Universal Robots URScript: etalement_vINIT.script

# UR5 - Protocole etalement cosmetique
# Genere automatiquement par ur5_etalement.py
# IMPORTANT : calibrer ROBOT_X_ORIGIN, ROBOT_Y_ORIGIN, ROBOT_Z_SURFACE avant execution

# --- Ancre globale du repere de travail ---
# P_ANCHOR_OLD : ancre nominale de la trajectoire originale (NE PAS MODIFIER)
# P_REF        : ancre cible. Modifier cette ligne pour relocaliser toute la zone d'etalement.
global P_ANCHOR_OLD = p[0.2,   -0.335, 0.05, 3.14159, 0.0, 0.0]
global P_REF        = p[-0.011, 0.6,   -0.3, 0.0, -3.1416, 0.0]


#TODO 5- Le nombre de lignes de code dans le script généré pour le robot UR5 dans UR5_etalementv6.py, est potentiellement trop élevé. Ce nombre de ligne de code dans le script est directement lié à la discretisation des cercles avec leur translation et la commande de force lors de chaque déplacement du robot UR5 sur le plan X-Y. Une option serait d'utiliser une fonction dans le robot UR5 pour réaliser des cercles avec translation sans l'utilisation de points avec la fonction movel tout en conservant en tout temps une commande pour 6N perpendiculaire au plan. Propose un plan pour réaliser ces fonctions dédiées. L'option des points de discrétisation doit demeurer. Il faut ajouter une option pour utiliser une fonction cercle+translation avec une sélection sous les figures.

# --- Vitesses (m/s) par phase ---
global V_APPROACH = 0.3
global V_CONTACT  = 0.05
global V_CIRC     = 0.0360
global V_RECT     = 0.0800
global V_INIT     = 0.5

# --- Accelerations (m/s^2) par phase ---
global A_DEFAULT  = 0.8
global A_INIT     = 1.2

# --- Facteurs multiplicateurs globaux ---
# 1.0 = nominal. Reduire SPEED_FACTOR pour mise au point.
global SPEED_FACTOR = 1.0
global ACCEL_FACTOR = 1.0

def T(p_orig):
  return pose_trans(P_REF, pose_trans(pose_inv(P_ANCHOR_OLD), p_orig))
end

def cycle_1():
  # --- Cycle 1 - Circulaire (0deg) ---
  movel(T(p[0.196464, -0.310607, 0.060000, 3.14159, 0.0, 0.0]), a=A_DEFAULT*ACCEL_FACTOR, v=V_APPROACH*SPEED_FACTOR)
  movel(T(p[0.196464, -0.310607, 0.050000, 3.14159, 0.0, 0.0]), a=A_DEFAULT*ACCEL_FACTOR, v=V_CONTACT*SPEED_FACTOR)
  force_mode(get_actual_tcp_pose(), [0, 0, 1, 0, 0, 0], [0, 0, -6.0, 0, 0, 0], 2, [0.002, 0.002, 0.04, 0.35, 0.35, 0.35])
  movel(T(p[0.198247, -0.304185, 0.050000, 3.14159, 0.0, 0.0]), a=A_DEFAULT*ACCEL_FACTOR, v=V_CIRC*SPEED_FACTOR, r=0.002)
  movel(T(p[0.206814, -0.307177, 0.050000, 3.14159, 0.0, 0.0]), a=A_DEFAULT*ACCEL_FACTOR, v=V_CIRC*SPEED_FACTOR, r=0.002)
  movel(T(p[0.205001, -0.315356, 0.050000, 3.14159, 0.0, 0.0]), a=A_DEFAULT*ACCEL_FACTOR, v=V_CIRC*SPEED_FACTOR, r=0.002)
  movel(T(p[0.199733, -0.312459, 0.050000, 3.14159, 0.0, 0.0]), a=A_DEFAULT*ACCEL_FACTOR, v=V_CIRC*SPEED_FACTOR, r=0.002)
  movel(T(p[0.206632, -0.307954, 0.050000, 3.14159, 0.0, 0.0]), a=A_DEFAULT*ACCEL_FACTOR, v=V_CIRC*SPEED_FACTOR, r=0.002)
  movel(T(p[0.211681, -0.315756, 0.050000, 3.14159, 0.0, 0.0]), a=A_DEFAULT*ACCEL_FACTOR, v=V_CIRC*SPEED_FACTOR, r=0.002)
  movel(T(p[0.205611, -0.319527, 0.050000, 3.14159, 0.0, 0.0]), a=A_DEFAULT*ACCEL_FACTOR, v=V_CIRC*SPEED_FACTOR, r=0.002)
  movel(T(p[0.205535, -0.313103, 0.050000, 3.14159, 0.0, 0.0]), a=A_DEFAULT*ACCEL_FACTOR, v=V_CIRC*SPEED_FACTOR, r=0.002)
  movel(T(p[0.214388, -0.314433, 0.050000, 3.14159, 0.0, 0.0]), a=A_DEFAULT*ACCEL_FACTOR, v=V_CIRC*SPEED_FACTOR, r=0.002)
  movel(T(p[0.213984, -0.323127, 0.050000, 3.14159, 0.0, 0.0]), a=A_DEFAULT*ACCEL_FACTOR, v=V_CIRC*SPEED_FACTOR, r=0.002)
  movel(T(p[0.208033, -0.321374, 0.050000, 3.14159, 0.0, 0.0]), a=A_DEFAULT*ACCEL_FACTOR, v=V_CIRC*SPEED_FACTOR, r=0.002)
  movel(T(p[0.213367, -0.316077, 0.050000, 3.14159, 0.0, 0.0]), a=A_DEFAULT*ACCEL_FACTOR, v=V_CIRC*SPEED_FACTOR, r=0.002)
  movel(T(p[0.220124, -0.322521, 0.050000, 3.14159, 0.0, 0.0]), a=A_DEFAULT*ACCEL_FACTOR, v=V_CIRC*SPEED_FACTOR, r=0.002)
  movel(T(p[0.215077, -0.328218, 0.050000, 3.14159, 0.0, 0.0]), a=A_DEFAULT*ACCEL_FACTOR, v=V_CIRC*SPEED_FACTOR, r=0.002)
  movel(T(p[0.212920, -0.322447, 0.050000, 3.14159, 0.0, 0.0]), a=A_DEFAULT*ACCEL_FACTOR, v=V_CIRC*SPEED_FACTOR, r=0.002)
  movel(T(p[0.221510, -0.321613, 0.050000, 3.14159, 0.0, 0.0]), a=A_DEFAULT*ACCEL_FACTOR, v=V_CIRC*SPEED_FACTOR, r=0.002)
  movel(T(p[0.223283, -0.330444, 0.050000, 3.14159, 0.0, 0.0]), a=A_DEFAULT*ACCEL_FACTOR, v=V_CIRC*SPEED_FACTOR, r=0.002)
  movel(T(p[0.216799, -0.330806, 0.050000, 3.14159, 0.0, 0.0]), a=A_DEFAULT*ACCEL_FACTOR, v=V_CIRC*SPEED_FACTOR, r=0.002)
  movel(T(p[0.220152, -0.324598, 0.050000, 3.14159, 0.0, 0.0]), a=A_DEFAULT*ACCEL_FACTOR, v=V_CIRC*SPEED_FACTOR, r=0.002)
  movel(T(p[0.228165, -0.329259, 0.050000, 3.14159, 0.0, 0.0]), a=A_DEFAULT*ACCEL_FACTOR, v=V_CIRC*SPEED_FACTOR, r=0.002)
  movel(T(p[0.224257, -0.340672, 0.050000, 3.14159, 0.0, 0.0]), a=A_DEFAULT*ACCEL_FACTOR, v=V_CIRC*SPEED_FACTOR, r=0.002)
  movel(T(p[0.224298, -0.337927, 0.050000, 3.14159, 0.0, 0.0]), a=A_DEFAULT*ACCEL_FACTOR, v=V_CIRC*SPEED_FACTOR, r=0.002)
  movel(T(p[0.210179, -0.336950, 0.050000, 3.14159, 0.0, 0.0]), a=A_DEFAULT*ACCEL_FACTOR, v=V_CIRC*SPEED_FACTOR, r=0.002)
  movel(T(p[0.216700, -0.335572, 0.050000, 3.14159, 0.0, 0.0]), a=A_DEFAULT*ACCEL_FACTOR, v=V_CIRC*SPEED_FACTOR, r=0.002)
  movel(T(p[0.214342, -0.342004, 0.050000, 3.14159, 0.0, 0.0]), a=A_DEFAULT*ACCEL_FACTOR, v=V_CIRC*SPEED_FACTOR, r=0.002)
  movel(T(p[0.205926, -0.338276, 0.050000, 3.14159, 0.0, 0.0]), a=A_DEFAULT*ACCEL_FACTOR, v=V_CIRC*SPEED_FACTOR, r=0.002)
  movel(T(p[0.208605, -0.330451, 0.050000, 3.14159, 0.0, 0.0]), a=A_DEFAULT*ACCEL_FACTOR, v=V_CIRC*SPEED_FACTOR, r=0.002)
  movel(T(p[0.213287, -0.334283, 0.050000, 3.14159, 0.0, 0.0]), a=A_DEFAULT*ACCEL_FACTOR, v=V_CIRC*SPEED_FACTOR, r=0.002)
  movel(T(p[0.206141, -0.337953, 0.050000, 3.14159, 0.0, 0.0]), a=A_DEFAULT*ACCEL_FACTOR, v=V_CIRC*SPEED_FACTOR, r=0.002)
  movel(T(p[0.201316, -0.330024, 0.050000, 3.14159, 0.0, 0.0]), a=A_DEFAULT*ACCEL_FACTOR, v=V_CIRC*SPEED_FACTOR, r=0.002)
  movel(T(p[0.207470, -0.326497, 0.050000, 3.14159, 0.0, 0.0]), a=A_DEFAULT*ACCEL_FACTOR, v=V_CIRC*SPEED_FACTOR, r=0.002)
  movel(T(p[0.207291, -0.332959, 0.050000, 3.14159, 0.0, 0.0]), a=A_DEFAULT*ACCEL_FACTOR, v=V_CIRC*SPEED_FACTOR, r=0.002)
  movel(T(p[0.198448, -0.331369, 0.050000, 3.14159, 0.0, 0.0]), a=A_DEFAULT*ACCEL_FACTOR, v=V_CIRC*SPEED_FACTOR, r=0.002)
  movel(T(p[0.199103, -0.322733, 0.050000, 3.14159, 0.0, 0.0]), a=A_DEFAULT*ACCEL_FACTOR, v=V_CIRC*SPEED_FACTOR, r=0.002)
  movel(T(p[0.204951, -0.324723, 0.050000, 3.14159, 0.0, 0.0]), a=A_DEFAULT*ACCEL_FACTOR, v=V_CIRC*SPEED_FACTOR, r=0.002)
  movel(T(p[0.199404, -0.329877, 0.050000, 3.14159, 0.0, 0.0]), a=A_DEFAULT*ACCEL_FACTOR, v=V_CIRC*SPEED_FACTOR, r=0.002)
  movel(T(p[0.192828, -0.323249, 0.050000, 3.14159, 0.0, 0.0]), a=A_DEFAULT*ACCEL_FACTOR, v=V_CIRC*SPEED_FACTOR, r=0.002)
  movel(T(p[0.198024, -0.317762, 0.050000, 3.14159, 0.0, 0.0]), a=A_DEFAULT*ACCEL_FACTOR, v=V_CIRC*SPEED_FACTOR, r=0.002)
  movel(T(p[0.199946, -0.323641, 0.050000, 3.14159, 0.0, 0.0]), a=A_DEFAULT*ACCEL_FACTOR, v=V_CIRC*SPEED_FACTOR, r=0.002)
  movel(T(p[0.191594, -0.323878, 0.050000, 3.14159, 0.0, 0.0]), a=A_DEFAULT*ACCEL_FACTOR, v=V_CIRC*SPEED_FACTOR, r=0.002)
  movel(T(p[0.184241, -0.319409, 0.050000, 3.14159, 0.0, 0.0]), a=A_DEFAULT*ACCEL_FACTOR, v=V_CIRC*SPEED_FACTOR, r=0.002)
  movel(T(p[0.184896, -0.325887, 0.050000, 3.14159, 0.0, 0.0]), a=A_DEFAULT*ACCEL_FACTOR, v=V_CIRC*SPEED_FACTOR, r=0.002)
  movel(T(p[0.192145, -0.331753, 0.050000, 3.14159, 0.0, 0.0]), a=A_DEFAULT*ACCEL_FACTOR, v=V_CIRC*SPEED_FACTOR, r=0.002)
  movel(T(p[0.187575, -0.338042, 0.050000, 3.14159, 0.0, 0.0]), a=A_DEFAULT*ACCEL_FACTOR, v=V_CIRC*SPEED_FACTOR, r=0.002)
  movel(T(p[0.184751, -0.332632, 0.050000, 3.14159, 0.0, 0.0]), a=A_DEFAULT*ACCEL_FACTOR, v=V_CIRC*SPEED_FACTOR, r=0.002)
  movel(T(p[0.193108, -0.331077, 0.050000, 3.14159, 0.0, 0.0]), a=A_DEFAULT*ACCEL_FACTOR, v=V_CIRC*SPEED_FACTOR, r=0.002)
  movel(T(p[0.195634, -0.339809, 0.050000, 3.14159, 0.0, 0.0]), a=A_DEFAULT*ACCEL_FACTOR, v=V_CIRC*SPEED_FACTOR, r=0.002)
  movel(T(p[0.189108, -0.340929, 0.050000, 3.14159, 0.0, 0.0]), a=A_DEFAULT*ACCEL_FACTOR, v=V_CIRC*SPEED_FACTOR, r=0.002)
  movel(T(p[0.191723, -0.334542, 0.050000, 3.14159, 0.0, 0.0]), a=A_DEFAULT*ACCEL_FACTOR, v=V_CIRC*SPEED_FACTOR, r=0.002)
  movel(T(p[0.200047, -0.338511, 0.050000, 3.14159, 0.0, 0.0]), a=A_DEFAULT*ACCEL_FACTOR, v=V_CIRC*SPEED_FACTOR, r=0.002)
  movel(T(p[0.197147, -0.346203, 0.050000, 3.14159, 0.0, 0.0]), a=A_DEFAULT*ACCEL_FACTOR, v=V_CIRC*SPEED_FACTOR, r=0.002)
  movel(T(p[0.192637, -0.342178, 0.050000, 3.14159, 0.0, 0.0]), a=A_DEFAULT*ACCEL_FACTOR, v=V_CIRC*SPEED_FACTOR, r=0.002)
  movel(T(p[0.199941, -0.338712, 0.050000, 3.14159, 0.0, 0.0]), a=A_DEFAULT*ACCEL_FACTOR, v=V_CIRC*SPEED_FACTOR, r=0.002)
  movel(T(p[0.204537, -0.346760, 0.050000, 3.14159, 0.0, 0.0]), a=A_DEFAULT*ACCEL_FACTOR, v=V_CIRC*SPEED_FACTOR, r=0.002)
  movel(T(p[0.198308, -0.350040, 0.050000, 3.14159, 0.0, 0.0]), a=A_DEFAULT*ACCEL_FACTOR, v=V_CIRC*SPEED_FACTOR, r=0.002)
  movel(T(p[0.198743, -0.343549, 0.050000, 3.14159, 0.0, 0.0]), a=A_DEFAULT*ACCEL_FACTOR, v=V_CIRC*SPEED_FACTOR, r=0.002)
  movel(T(p[0.207568, -0.345396, 0.050000, 3.14159, 0.0, 0.0]), a=A_DEFAULT*ACCEL_FACTOR, v=V_CIRC*SPEED_FACTOR, r=0.002)
  movel(T(p[0.206662, -0.353966, 0.050000, 3.14159, 0.0, 0.0]), a=A_DEFAULT*ACCEL_FACTOR, v=V_CIRC*SPEED_FACTOR, r=0.002)
  movel(T(p[0.210965, -0.358063, 0.050000, 3.14159, 0.0, 0.0]), a=A_DEFAULT*ACCEL_FACTOR, v=V_CIRC*SPEED_FACTOR, r=0.002)
  movel(T(p[0.197831, -0.356868, 0.050000, 3.14159, 0.0, 0.0]), a=A_DEFAULT*ACCEL_FACTOR, v=V_CIRC*SPEED_FACTOR, r=0.002)
  movel(T(p[0.197313, -0.354239, 0.050000, 3.14159, 0.0, 0.0]), a=A_DEFAULT*ACCEL_FACTOR, v=V_CIRC*SPEED_FACTOR, r=0.002)
  movel(T(p[0.197882, -0.360567, 0.050000, 3.14159, 0.0, 0.0]), a=A_DEFAULT*ACCEL_FACTOR, v=V_CIRC*SPEED_FACTOR, r=0.002)
  movel(T(p[0.189034, -0.359736, 0.050000, 3.14159, 0.0, 0.0]), a=A_DEFAULT*ACCEL_FACTOR, v=V_CIRC*SPEED_FACTOR, r=0.002)
  movel(T(p[0.188944, -0.350957, 0.050000, 3.14159, 0.0, 0.0]), a=A_DEFAULT*ACCEL_FACTOR, v=V_CIRC*SPEED_FACTOR, r=0.002)
  movel(T(p[0.195069, -0.352240, 0.050000, 3.14159, 0.0, 0.0]), a=A_DEFAULT*ACCEL_FACTOR, v=V_CIRC*SPEED_FACTOR, r=0.002)
  movel(T(p[0.190166, -0.357795, 0.050000, 3.14159, 0.0, 0.0]), a=A_DEFAULT*ACCEL_FACTOR, v=V_CIRC*SPEED_FACTOR, r=0.002)
  movel(T(p[0.183077, -0.351727, 0.050000, 3.14159, 0.0, 0.0]), a=A_DEFAULT*ACCEL_FACTOR, v=V_CIRC*SPEED_FACTOR, r=0.002)
  movel(T(p[0.187816, -0.345635, 0.050000, 3.14159, 0.0, 0.0]), a=A_DEFAULT*ACCEL_FACTOR, v=V_CIRC*SPEED_FACTOR, r=0.002)
  movel(T(p[0.190418, -0.351174, 0.050000, 3.14159, 0.0, 0.0]), a=A_DEFAULT*ACCEL_FACTOR, v=V_CIRC*SPEED_FACTOR, r=0.002)
  movel(T(p[0.181973, -0.352487, 0.050000, 3.14159, 0.0, 0.0]), a=A_DEFAULT*ACCEL_FACTOR, v=V_CIRC*SPEED_FACTOR, r=0.002)
  movel(T(p[0.179702, -0.343713, 0.050000, 3.14159, 0.0, 0.0]), a=A_DEFAULT*ACCEL_FACTOR, v=V_CIRC*SPEED_FACTOR, r=0.002)
  movel(T(p[0.186221, -0.342851, 0.050000, 3.14159, 0.0, 0.0]), a=A_DEFAULT*ACCEL_FACTOR, v=V_CIRC*SPEED_FACTOR, r=0.002)
  movel(T(p[0.183355, -0.349185, 0.050000, 3.14159, 0.0, 0.0]), a=A_DEFAULT*ACCEL_FACTOR, v=V_CIRC*SPEED_FACTOR, r=0.002)
  movel(T(p[0.175128, -0.344978, 0.050000, 3.14159, 0.0, 0.0]), a=A_DEFAULT*ACCEL_FACTOR, v=V_CIRC*SPEED_FACTOR, r=0.002)
  movel(T(p[0.178246, -0.337425, 0.050000, 3.14159, 0.0, 0.0]), a=A_DEFAULT*ACCEL_FACTOR, v=V_CIRC*SPEED_FACTOR, r=0.002)
  movel(T(p[0.182578, -0.341638, 0.050000, 3.14159, 0.0, 0.0]), a=A_DEFAULT*ACCEL_FACTOR, v=V_CIRC*SPEED_FACTOR, r=0.002)
  movel(T(p[0.175123, -0.344896, 0.050000, 3.14159, 0.0, 0.0]), a=A_DEFAULT*ACCEL_FACTOR, v=V_CIRC*SPEED_FACTOR, r=0.002)
  movel(T(p[0.171025, -0.336323, 0.050000, 3.14159, 0.0, 0.0]), a=A_DEFAULT*ACCEL_FACTOR, v=V_CIRC*SPEED_FACTOR, r=0.002)
  movel(T(p[0.177378, -0.333966, 0.050000, 3.14159, 0.0, 0.0]), a=A_DEFAULT*ACCEL_FACTOR, v=V_CIRC*SPEED_FACTOR, r=0.002)
  movel(T(p[0.176172, -0.340413, 0.050000, 3.14159, 0.0, 0.0]), a=A_DEFAULT*ACCEL_FACTOR, v=V_CIRC*SPEED_FACTOR, r=0.002)
  movel(T(p[0.167489, -0.337986, 0.050000, 3.14159, 0.0, 0.0]), a=A_DEFAULT*ACCEL_FACTOR, v=V_CIRC*SPEED_FACTOR, r=0.002)
  end_force_mode()
  movel(T(p[0.168180, -0.338891, 0.060000, 3.14159, 0.0, 0.0]), a=A_DEFAULT*ACCEL_FACTOR, v=V_APPROACH*SPEED_FACTOR)
end

def cycle_2():
  # --- Cycle 2 - Circulaire (90deg) ---
  movel(T(p[0.175251, -0.338891, 0.060000, 3.14159, 0.0, 0.0]), a=A_DEFAULT*ACCEL_FACTOR, v=V_APPROACH*SPEED_FACTOR)
  movel(T(p[0.175251, -0.338891, 0.050000, 3.14159, 0.0, 0.0]), a=A_DEFAULT*ACCEL_FACTOR, v=V_CONTACT*SPEED_FACTOR)
  force_mode(get_actual_tcp_pose(), [0, 0, 1, 0, 0, 0], [0, 0, -6.0, 0, 0, 0], 2, [0.002, 0.002, 0.04, 0.35, 0.35, 0.35])
  movel(T(p[0.168830, -0.337108, 0.050000, 3.14159, 0.0, 0.0]), a=A_DEFAULT*ACCEL_FACTOR, v=V_CIRC*SPEED_FACTOR, r=0.002)
  movel(T(p[0.171822, -0.328542, 0.050000, 3.14159, 0.0, 0.0]), a=A_DEFAULT*ACCEL_FACTOR, v=V_CIRC*SPEED_FACTOR, r=0.002)
  movel(T(p[0.180001, -0.330354, 0.050000, 3.14159, 0.0, 0.0]), a=A_DEFAULT*ACCEL_FACTOR, v=V_CIRC*SPEED_FACTOR, r=0.002)
  movel(T(p[0.177104, -0.335623, 0.050000, 3.14159, 0.0, 0.0]), a=A_DEFAULT*ACCEL_FACTOR, v=V_CIRC*SPEED_FACTOR, r=0.002)
  movel(T(p[0.172599, -0.328723, 0.050000, 3.14159, 0.0, 0.0]), a=A_DEFAULT*ACCEL_FACTOR, v=V_CIRC*SPEED_FACTOR, r=0.002)
  movel(T(p[0.180400, -0.323674, 0.050000, 3.14159, 0.0, 0.0]), a=A_DEFAULT*ACCEL_FACTOR, v=V_CIRC*SPEED_FACTOR, r=0.002)
  movel(T(p[0.184171, -0.329744, 0.050000, 3.14159, 0.0, 0.0]), a=A_DEFAULT*ACCEL_FACTOR, v=V_CIRC*SPEED_FACTOR, r=0.002)
  movel(T(p[0.177747, -0.329820, 0.050000, 3.14159, 0.0, 0.0]), a=A_DEFAULT*ACCEL_FACTOR, v=V_CIRC*SPEED_FACTOR, r=0.002)
  movel(T(p[0.179078, -0.320967, 0.050000, 3.14159, 0.0, 0.0]), a=A_DEFAULT*ACCEL_FACTOR, v=V_CIRC*SPEED_FACTOR, r=0.002)
  movel(T(p[0.187771, -0.321372, 0.050000, 3.14159, 0.0, 0.0]), a=A_DEFAULT*ACCEL_FACTOR, v=V_CIRC*SPEED_FACTOR, r=0.002)
  movel(T(p[0.186018, -0.327322, 0.050000, 3.14159, 0.0, 0.0]), a=A_DEFAULT*ACCEL_FACTOR, v=V_CIRC*SPEED_FACTOR, r=0.002)
  movel(T(p[0.180721, -0.321988, 0.050000, 3.14159, 0.0, 0.0]), a=A_DEFAULT*ACCEL_FACTOR, v=V_CIRC*SPEED_FACTOR, r=0.002)
  movel(T(p[0.187165, -0.315232, 0.050000, 3.14159, 0.0, 0.0]), a=A_DEFAULT*ACCEL_FACTOR, v=V_CIRC*SPEED_FACTOR, r=0.002)
  movel(T(p[0.192862, -0.320278, 0.050000, 3.14159, 0.0, 0.0]), a=A_DEFAULT*ACCEL_FACTOR, v=V_CIRC*SPEED_FACTOR, r=0.002)
  movel(T(p[0.187092, -0.322436, 0.050000, 3.14159, 0.0, 0.0]), a=A_DEFAULT*ACCEL_FACTOR, v=V_CIRC*SPEED_FACTOR, r=0.002)
  movel(T(p[0.186258, -0.313845, 0.050000, 3.14159, 0.0, 0.0]), a=A_DEFAULT*ACCEL_FACTOR, v=V_CIRC*SPEED_FACTOR, r=0.002)
  movel(T(p[0.195089, -0.312072, 0.050000, 3.14159, 0.0, 0.0]), a=A_DEFAULT*ACCEL_FACTOR, v=V_CIRC*SPEED_FACTOR, r=0.002)
  movel(T(p[0.195450, -0.318556, 0.050000, 3.14159, 0.0, 0.0]), a=A_DEFAULT*ACCEL_FACTOR, v=V_CIRC*SPEED_FACTOR, r=0.002)
  movel(T(p[0.189243, -0.315204, 0.050000, 3.14159, 0.0, 0.0]), a=A_DEFAULT*ACCEL_FACTOR, v=V_CIRC*SPEED_FACTOR, r=0.002)
  movel(T(p[0.193904, -0.307191, 0.050000, 3.14159, 0.0, 0.0]), a=A_DEFAULT*ACCEL_FACTOR, v=V_CIRC*SPEED_FACTOR, r=0.002)
  movel(T(p[0.205317, -0.311098, 0.050000, 3.14159, 0.0, 0.0]), a=A_DEFAULT*ACCEL_FACTOR, v=V_CIRC*SPEED_FACTOR, r=0.002)
  movel(T(p[0.202572, -0.311057, 0.050000, 3.14159, 0.0, 0.0]), a=A_DEFAULT*ACCEL_FACTOR, v=V_CIRC*SPEED_FACTOR, r=0.002)
  movel(T(p[0.201595, -0.325177, 0.050000, 3.14159, 0.0, 0.0]), a=A_DEFAULT*ACCEL_FACTOR, v=V_CIRC*SPEED_FACTOR, r=0.002)
  movel(T(p[0.200216, -0.318655, 0.050000, 3.14159, 0.0, 0.0]), a=A_DEFAULT*ACCEL_FACTOR, v=V_CIRC*SPEED_FACTOR, r=0.002)
  movel(T(p[0.206648, -0.321014, 0.050000, 3.14159, 0.0, 0.0]), a=A_DEFAULT*ACCEL_FACTOR, v=V_CIRC*SPEED_FACTOR, r=0.002)
  movel(T(p[0.202920, -0.329430, 0.050000, 3.14159, 0.0, 0.0]), a=A_DEFAULT*ACCEL_FACTOR, v=V_CIRC*SPEED_FACTOR, r=0.002)
  movel(T(p[0.195096, -0.326750, 0.050000, 3.14159, 0.0, 0.0]), a=A_DEFAULT*ACCEL_FACTOR, v=V_CIRC*SPEED_FACTOR, r=0.002)
  movel(T(p[0.198928, -0.322069, 0.050000, 3.14159, 0.0, 0.0]), a=A_DEFAULT*ACCEL_FACTOR, v=V_CIRC*SPEED_FACTOR, r=0.002)
  movel(T(p[0.202597, -0.329214, 0.050000, 3.14159, 0.0, 0.0]), a=A_DEFAULT*ACCEL_FACTOR, v=V_CIRC*SPEED_FACTOR, r=0.002)
  movel(T(p[0.194669, -0.334039, 0.050000, 3.14159, 0.0, 0.0]), a=A_DEFAULT*ACCEL_FACTOR, v=V_CIRC*SPEED_FACTOR, r=0.002)
  movel(T(p[0.191141, -0.327885, 0.050000, 3.14159, 0.0, 0.0]), a=A_DEFAULT*ACCEL_FACTOR, v=V_CIRC*SPEED_FACTOR, r=0.002)
  movel(T(p[0.197604, -0.328064, 0.050000, 3.14159, 0.0, 0.0]), a=A_DEFAULT*ACCEL_FACTOR, v=V_CIRC*SPEED_FACTOR, r=0.002)
  movel(T(p[0.196014, -0.336907, 0.050000, 3.14159, 0.0, 0.0]), a=A_DEFAULT*ACCEL_FACTOR, v=V_CIRC*SPEED_FACTOR, r=0.002)
  movel(T(p[0.187378, -0.336252, 0.050000, 3.14159, 0.0, 0.0]), a=A_DEFAULT*ACCEL_FACTOR, v=V_CIRC*SPEED_FACTOR, r=0.002)
  movel(T(p[0.189368, -0.330404, 0.050000, 3.14159, 0.0, 0.0]), a=A_DEFAULT*ACCEL_FACTOR, v=V_CIRC*SPEED_FACTOR, r=0.002)
  movel(T(p[0.194522, -0.335951, 0.050000, 3.14159, 0.0, 0.0]), a=A_DEFAULT*ACCEL_FACTOR, v=V_CIRC*SPEED_FACTOR, r=0.002)
  movel(T(p[0.187894, -0.342528, 0.050000, 3.14159, 0.0, 0.0]), a=A_DEFAULT*ACCEL_FACTOR, v=V_CIRC*SPEED_FACTOR, r=0.002)
  movel(T(p[0.182406, -0.337332, 0.050000, 3.14159, 0.0, 0.0]), a=A_DEFAULT*ACCEL_FACTOR, v=V_CIRC*SPEED_FACTOR, r=0.002)
  movel(T(p[0.188285, -0.335410, 0.050000, 3.14159, 0.0, 0.0]), a=A_DEFAULT*ACCEL_FACTOR, v=V_CIRC*SPEED_FACTOR, r=0.002)
  movel(T(p[0.188522, -0.343761, 0.050000, 3.14159, 0.0, 0.0]), a=A_DEFAULT*ACCEL_FACTOR, v=V_CIRC*SPEED_FACTOR, r=0.002)
  movel(T(p[0.184054, -0.351115, 0.050000, 3.14159, 0.0, 0.0]), a=A_DEFAULT*ACCEL_FACTOR, v=V_CIRC*SPEED_FACTOR, r=0.002)
  movel(T(p[0.190532, -0.350459, 0.050000, 3.14159, 0.0, 0.0]), a=A_DEFAULT*ACCEL_FACTOR, v=V_CIRC*SPEED_FACTOR, r=0.002)
  movel(T(p[0.196398, -0.343210, 0.050000, 3.14159, 0.0, 0.0]), a=A_DEFAULT*ACCEL_FACTOR, v=V_CIRC*SPEED_FACTOR, r=0.002)
  movel(T(p[0.202686, -0.347780, 0.050000, 3.14159, 0.0, 0.0]), a=A_DEFAULT*ACCEL_FACTOR, v=V_CIRC*SPEED_FACTOR, r=0.002)
  movel(T(p[0.197277, -0.350604, 0.050000, 3.14159, 0.0, 0.0]), a=A_DEFAULT*ACCEL_FACTOR, v=V_CIRC*SPEED_FACTOR, r=0.002)
  movel(T(p[0.195721, -0.342248, 0.050000, 3.14159, 0.0, 0.0]), a=A_DEFAULT*ACCEL_FACTOR, v=V_CIRC*SPEED_FACTOR, r=0.002)
  movel(T(p[0.204454, -0.339722, 0.050000, 3.14159, 0.0, 0.0]), a=A_DEFAULT*ACCEL_FACTOR, v=V_CIRC*SPEED_FACTOR, r=0.002)
  movel(T(p[0.205574, -0.346247, 0.050000, 3.14159, 0.0, 0.0]), a=A_DEFAULT*ACCEL_FACTOR, v=V_CIRC*SPEED_FACTOR, r=0.002)
  movel(T(p[0.199187, -0.343633, 0.050000, 3.14159, 0.0, 0.0]), a=A_DEFAULT*ACCEL_FACTOR, v=V_CIRC*SPEED_FACTOR, r=0.002)
  movel(T(p[0.203156, -0.335308, 0.050000, 3.14159, 0.0, 0.0]), a=A_DEFAULT*ACCEL_FACTOR, v=V_CIRC*SPEED_FACTOR, r=0.002)
  movel(T(p[0.210848, -0.338209, 0.050000, 3.14159, 0.0, 0.0]), a=A_DEFAULT*ACCEL_FACTOR, v=V_CIRC*SPEED_FACTOR, r=0.002)
  movel(T(p[0.206823, -0.342718, 0.050000, 3.14159, 0.0, 0.0]), a=A_DEFAULT*ACCEL_FACTOR, v=V_CIRC*SPEED_FACTOR, r=0.002)
  movel(T(p[0.203357, -0.335414, 0.050000, 3.14159, 0.0, 0.0]), a=A_DEFAULT*ACCEL_FACTOR, v=V_CIRC*SPEED_FACTOR, r=0.002)
  movel(T(p[0.211404, -0.330819, 0.050000, 3.14159, 0.0, 0.0]), a=A_DEFAULT*ACCEL_FACTOR, v=V_CIRC*SPEED_FACTOR, r=0.002)
  movel(T(p[0.214684, -0.337047, 0.050000, 3.14159, 0.0, 0.0]), a=A_DEFAULT*ACCEL_FACTOR, v=V_CIRC*SPEED_FACTOR, r=0.002)
  movel(T(p[0.208193, -0.336612, 0.050000, 3.14159, 0.0, 0.0]), a=A_DEFAULT*ACCEL_FACTOR, v=V_CIRC*SPEED_FACTOR, r=0.002)
  movel(T(p[0.210040, -0.327787, 0.050000, 3.14159, 0.0, 0.0]), a=A_DEFAULT*ACCEL_FACTOR, v=V_CIRC*SPEED_FACTOR, r=0.002)
  movel(T(p[0.218611, -0.328693, 0.050000, 3.14159, 0.0, 0.0]), a=A_DEFAULT*ACCEL_FACTOR, v=V_CIRC*SPEED_FACTOR, r=0.002)
  movel(T(p[0.222707, -0.324390, 0.050000, 3.14159, 0.0, 0.0]), a=A_DEFAULT*ACCEL_FACTOR, v=V_CIRC*SPEED_FACTOR, r=0.002)
  movel(T(p[0.221512, -0.337524, 0.050000, 3.14159, 0.0, 0.0]), a=A_DEFAULT*ACCEL_FACTOR, v=V_CIRC*SPEED_FACTOR, r=0.002)
  movel(T(p[0.218884, -0.338042, 0.050000, 3.14159, 0.0, 0.0]), a=A_DEFAULT*ACCEL_FACTOR, v=V_CIRC*SPEED_FACTOR, r=0.002)
  movel(T(p[0.225211, -0.337474, 0.050000, 3.14159, 0.0, 0.0]), a=A_DEFAULT*ACCEL_FACTOR, v=V_CIRC*SPEED_FACTOR, r=0.002)
  movel(T(p[0.224381, -0.346321, 0.050000, 3.14159, 0.0, 0.0]), a=A_DEFAULT*ACCEL_FACTOR, v=V_CIRC*SPEED_FACTOR, r=0.002)
  movel(T(p[0.215602, -0.346412, 0.050000, 3.14159, 0.0, 0.0]), a=A_DEFAULT*ACCEL_FACTOR, v=V_CIRC*SPEED_FACTOR, r=0.002)
  movel(T(p[0.216885, -0.340286, 0.050000, 3.14159, 0.0, 0.0]), a=A_DEFAULT*ACCEL_FACTOR, v=V_CIRC*SPEED_FACTOR, r=0.002)
  movel(T(p[0.222440, -0.345189, 0.050000, 3.14159, 0.0, 0.0]), a=A_DEFAULT*ACCEL_FACTOR, v=V_CIRC*SPEED_FACTOR, r=0.002)
  movel(T(p[0.216372, -0.352279, 0.050000, 3.14159, 0.0, 0.0]), a=A_DEFAULT*ACCEL_FACTOR, v=V_CIRC*SPEED_FACTOR, r=0.002)
  movel(T(p[0.210279, -0.347539, 0.050000, 3.14159, 0.0, 0.0]), a=A_DEFAULT*ACCEL_FACTOR, v=V_CIRC*SPEED_FACTOR, r=0.002)
  movel(T(p[0.215819, -0.344937, 0.050000, 3.14159, 0.0, 0.0]), a=A_DEFAULT*ACCEL_FACTOR, v=V_CIRC*SPEED_FACTOR, r=0.002)
  movel(T(p[0.217132, -0.353382, 0.050000, 3.14159, 0.0, 0.0]), a=A_DEFAULT*ACCEL_FACTOR, v=V_CIRC*SPEED_FACTOR, r=0.002)
  movel(T(p[0.208357, -0.355653, 0.050000, 3.14159, 0.0, 0.0]), a=A_DEFAULT*ACCEL_FACTOR, v=V_CIRC*SPEED_FACTOR, r=0.002)
  movel(T(p[0.207495, -0.349134, 0.050000, 3.14159, 0.0, 0.0]), a=A_DEFAULT*ACCEL_FACTOR, v=V_CIRC*SPEED_FACTOR, r=0.002)
  movel(T(p[0.213830, -0.352001, 0.050000, 3.14159, 0.0, 0.0]), a=A_DEFAULT*ACCEL_FACTOR, v=V_CIRC*SPEED_FACTOR, r=0.002)
  movel(T(p[0.209622, -0.360227, 0.050000, 3.14159, 0.0, 0.0]), a=A_DEFAULT*ACCEL_FACTOR, v=V_CIRC*SPEED_FACTOR, r=0.002)
  movel(T(p[0.202070, -0.357109, 0.050000, 3.14159, 0.0, 0.0]), a=A_DEFAULT*ACCEL_FACTOR, v=V_CIRC*SPEED_FACTOR, r=0.002)
  movel(T(p[0.206283, -0.352778, 0.050000, 3.14159, 0.0, 0.0]), a=A_DEFAULT*ACCEL_FACTOR, v=V_CIRC*SPEED_FACTOR, r=0.002)
  movel(T(p[0.209540, -0.360233, 0.050000, 3.14159, 0.0, 0.0]), a=A_DEFAULT*ACCEL_FACTOR, v=V_CIRC*SPEED_FACTOR, r=0.002)
  movel(T(p[0.200968, -0.364330, 0.050000, 3.14159, 0.0, 0.0]), a=A_DEFAULT*ACCEL_FACTOR, v=V_CIRC*SPEED_FACTOR, r=0.002)
  movel(T(p[0.198611, -0.357978, 0.050000, 3.14159, 0.0, 0.0]), a=A_DEFAULT*ACCEL_FACTOR, v=V_CIRC*SPEED_FACTOR, r=0.002)
  movel(T(p[0.205057, -0.359183, 0.050000, 3.14159, 0.0, 0.0]), a=A_DEFAULT*ACCEL_FACTOR, v=V_CIRC*SPEED_FACTOR, r=0.002)
  movel(T(p[0.202631, -0.367866, 0.050000, 3.14159, 0.0, 0.0]), a=A_DEFAULT*ACCEL_FACTOR, v=V_CIRC*SPEED_FACTOR, r=0.002)
  end_force_mode()
  movel(T(p[0.203536, -0.367175, 0.060000, 3.14159, 0.0, 0.0]), a=A_DEFAULT*ACCEL_FACTOR, v=V_APPROACH*SPEED_FACTOR)
end

def cycle_3():
  # --- Cycle 3 - Circulaire (0deg) ---
  movel(T(p[0.196464, -0.310607, 0.060000, 3.14159, 0.0, 0.0]), a=A_DEFAULT*ACCEL_FACTOR, v=V_APPROACH*SPEED_FACTOR)
  movel(T(p[0.196464, -0.310607, 0.050000, 3.14159, 0.0, 0.0]), a=A_DEFAULT*ACCEL_FACTOR, v=V_CONTACT*SPEED_FACTOR)
  force_mode(get_actual_tcp_pose(), [0, 0, 1, 0, 0, 0], [0, 0, -6.0, 0, 0, 0], 2, [0.002, 0.002, 0.04, 0.35, 0.35, 0.35])
  movel(T(p[0.198247, -0.304185, 0.050000, 3.14159, 0.0, 0.0]), a=A_DEFAULT*ACCEL_FACTOR, v=V_CIRC*SPEED_FACTOR, r=0.002)
  movel(T(p[0.206814, -0.307177, 0.050000, 3.14159, 0.0, 0.0]), a=A_DEFAULT*ACCEL_FACTOR, v=V_CIRC*SPEED_FACTOR, r=0.002)
  movel(T(p[0.205001, -0.315356, 0.050000, 3.14159, 0.0, 0.0]), a=A_DEFAULT*ACCEL_FACTOR, v=V_CIRC*SPEED_FACTOR, r=0.002)
  movel(T(p[0.199733, -0.312459, 0.050000, 3.14159, 0.0, 0.0]), a=A_DEFAULT*ACCEL_FACTOR, v=V_CIRC*SPEED_FACTOR, r=0.002)
  movel(T(p[0.206632, -0.307954, 0.050000, 3.14159, 0.0, 0.0]), a=A_DEFAULT*ACCEL_FACTOR, v=V_CIRC*SPEED_FACTOR, r=0.002)
  movel(T(p[0.211681, -0.315756, 0.050000, 3.14159, 0.0, 0.0]), a=A_DEFAULT*ACCEL_FACTOR, v=V_CIRC*SPEED_FACTOR, r=0.002)
  movel(T(p[0.205611, -0.319527, 0.050000, 3.14159, 0.0, 0.0]), a=A_DEFAULT*ACCEL_FACTOR, v=V_CIRC*SPEED_FACTOR, r=0.002)
  movel(T(p[0.205535, -0.313103, 0.050000, 3.14159, 0.0, 0.0]), a=A_DEFAULT*ACCEL_FACTOR, v=V_CIRC*SPEED_FACTOR, r=0.002)
  movel(T(p[0.214388, -0.314433, 0.050000, 3.14159, 0.0, 0.0]), a=A_DEFAULT*ACCEL_FACTOR, v=V_CIRC*SPEED_FACTOR, r=0.002)
  movel(T(p[0.213984, -0.323127, 0.050000, 3.14159, 0.0, 0.0]), a=A_DEFAULT*ACCEL_FACTOR, v=V_CIRC*SPEED_FACTOR, r=0.002)
  movel(T(p[0.208033, -0.321374, 0.050000, 3.14159, 0.0, 0.0]), a=A_DEFAULT*ACCEL_FACTOR, v=V_CIRC*SPEED_FACTOR, r=0.002)
  movel(T(p[0.213367, -0.316077, 0.050000, 3.14159, 0.0, 0.0]), a=A_DEFAULT*ACCEL_FACTOR, v=V_CIRC*SPEED_FACTOR, r=0.002)
  movel(T(p[0.220124, -0.322521, 0.050000, 3.14159, 0.0, 0.0]), a=A_DEFAULT*ACCEL_FACTOR, v=V_CIRC*SPEED_FACTOR, r=0.002)
  movel(T(p[0.215077, -0.328218, 0.050000, 3.14159, 0.0, 0.0]), a=A_DEFAULT*ACCEL_FACTOR, v=V_CIRC*SPEED_FACTOR, r=0.002)
  movel(T(p[0.212920, -0.322447, 0.050000, 3.14159, 0.0, 0.0]), a=A_DEFAULT*ACCEL_FACTOR, v=V_CIRC*SPEED_FACTOR, r=0.002)
  movel(T(p[0.221510, -0.321613, 0.050000, 3.14159, 0.0, 0.0]), a=A_DEFAULT*ACCEL_FACTOR, v=V_CIRC*SPEED_FACTOR, r=0.002)
  movel(T(p[0.223283, -0.330444, 0.050000, 3.14159, 0.0, 0.0]), a=A_DEFAULT*ACCEL_FACTOR, v=V_CIRC*SPEED_FACTOR, r=0.002)
  movel(T(p[0.216799, -0.330806, 0.050000, 3.14159, 0.0, 0.0]), a=A_DEFAULT*ACCEL_FACTOR, v=V_CIRC*SPEED_FACTOR, r=0.002)
  movel(T(p[0.220152, -0.324598, 0.050000, 3.14159, 0.0, 0.0]), a=A_DEFAULT*ACCEL_FACTOR, v=V_CIRC*SPEED_FACTOR, r=0.002)
  movel(T(p[0.228165, -0.329259, 0.050000, 3.14159, 0.0, 0.0]), a=A_DEFAULT*ACCEL_FACTOR, v=V_CIRC*SPEED_FACTOR, r=0.002)
  movel(T(p[0.224257, -0.340672, 0.050000, 3.14159, 0.0, 0.0]), a=A_DEFAULT*ACCEL_FACTOR, v=V_CIRC*SPEED_FACTOR, r=0.002)
  movel(T(p[0.224298, -0.337927, 0.050000, 3.14159, 0.0, 0.0]), a=A_DEFAULT*ACCEL_FACTOR, v=V_CIRC*SPEED_FACTOR, r=0.002)
  movel(T(p[0.210179, -0.336950, 0.050000, 3.14159, 0.0, 0.0]), a=A_DEFAULT*ACCEL_FACTOR, v=V_CIRC*SPEED_FACTOR, r=0.002)
  movel(T(p[0.216700, -0.335572, 0.050000, 3.14159, 0.0, 0.0]), a=A_DEFAULT*ACCEL_FACTOR, v=V_CIRC*SPEED_FACTOR, r=0.002)
  movel(T(p[0.214342, -0.342004, 0.050000, 3.14159, 0.0, 0.0]), a=A_DEFAULT*ACCEL_FACTOR, v=V_CIRC*SPEED_FACTOR, r=0.002)
  movel(T(p[0.205926, -0.338276, 0.050000, 3.14159, 0.0, 0.0]), a=A_DEFAULT*ACCEL_FACTOR, v=V_CIRC*SPEED_FACTOR, r=0.002)
  movel(T(p[0.208605, -0.330451, 0.050000, 3.14159, 0.0, 0.0]), a=A_DEFAULT*ACCEL_FACTOR, v=V_CIRC*SPEED_FACTOR, r=0.002)
  movel(T(p[0.213287, -0.334283, 0.050000, 3.14159, 0.0, 0.0]), a=A_DEFAULT*ACCEL_FACTOR, v=V_CIRC*SPEED_FACTOR, r=0.002)
  movel(T(p[0.206141, -0.337953, 0.050000, 3.14159, 0.0, 0.0]), a=A_DEFAULT*ACCEL_FACTOR, v=V_CIRC*SPEED_FACTOR, r=0.002)
  movel(T(p[0.201316, -0.330024, 0.050000, 3.14159, 0.0, 0.0]), a=A_DEFAULT*ACCEL_FACTOR, v=V_CIRC*SPEED_FACTOR, r=0.002)
  movel(T(p[0.207470, -0.326497, 0.050000, 3.14159, 0.0, 0.0]), a=A_DEFAULT*ACCEL_FACTOR, v=V_CIRC*SPEED_FACTOR, r=0.002)
  movel(T(p[0.207291, -0.332959, 0.050000, 3.14159, 0.0, 0.0]), a=A_DEFAULT*ACCEL_FACTOR, v=V_CIRC*SPEED_FACTOR, r=0.002)
  movel(T(p[0.198448, -0.331369, 0.050000, 3.14159, 0.0, 0.0]), a=A_DEFAULT*ACCEL_FACTOR, v=V_CIRC*SPEED_FACTOR, r=0.002)
  movel(T(p[0.199103, -0.322733, 0.050000, 3.14159, 0.0, 0.0]), a=A_DEFAULT*ACCEL_FACTOR, v=V_CIRC*SPEED_FACTOR, r=0.002)
  movel(T(p[0.204951, -0.324723, 0.050000, 3.14159, 0.0, 0.0]), a=A_DEFAULT*ACCEL_FACTOR, v=V_CIRC*SPEED_FACTOR, r=0.002)
  movel(T(p[0.199404, -0.329877, 0.050000, 3.14159, 0.0, 0.0]), a=A_DEFAULT*ACCEL_FACTOR, v=V_CIRC*SPEED_FACTOR, r=0.002)
  movel(T(p[0.192828, -0.323249, 0.050000, 3.14159, 0.0, 0.0]), a=A_DEFAULT*ACCEL_FACTOR, v=V_CIRC*SPEED_FACTOR, r=0.002)
  movel(T(p[0.198024, -0.317762, 0.050000, 3.14159, 0.0, 0.0]), a=A_DEFAULT*ACCEL_FACTOR, v=V_CIRC*SPEED_FACTOR, r=0.002)
  movel(T(p[0.199946, -0.323641, 0.050000, 3.14159, 0.0, 0.0]), a=A_DEFAULT*ACCEL_FACTOR, v=V_CIRC*SPEED_FACTOR, r=0.002)
  movel(T(p[0.191594, -0.323878, 0.050000, 3.14159, 0.0, 0.0]), a=A_DEFAULT*ACCEL_FACTOR, v=V_CIRC*SPEED_FACTOR, r=0.002)
  movel(T(p[0.184241, -0.319409, 0.050000, 3.14159, 0.0, 0.0]), a=A_DEFAULT*ACCEL_FACTOR, v=V_CIRC*SPEED_FACTOR, r=0.002)
  movel(T(p[0.184896, -0.325887, 0.050000, 3.14159, 0.0, 0.0]), a=A_DEFAULT*ACCEL_FACTOR, v=V_CIRC*SPEED_FACTOR, r=0.002)
  movel(T(p[0.192145, -0.331753, 0.050000, 3.14159, 0.0, 0.0]), a=A_DEFAULT*ACCEL_FACTOR, v=V_CIRC*SPEED_FACTOR, r=0.002)
  movel(T(p[0.187575, -0.338042, 0.050000, 3.14159, 0.0, 0.0]), a=A_DEFAULT*ACCEL_FACTOR, v=V_CIRC*SPEED_FACTOR, r=0.002)
  movel(T(p[0.184751, -0.332632, 0.050000, 3.14159, 0.0, 0.0]), a=A_DEFAULT*ACCEL_FACTOR, v=V_CIRC*SPEED_FACTOR, r=0.002)
  movel(T(p[0.193108, -0.331077, 0.050000, 3.14159, 0.0, 0.0]), a=A_DEFAULT*ACCEL_FACTOR, v=V_CIRC*SPEED_FACTOR, r=0.002)
  movel(T(p[0.195634, -0.339809, 0.050000, 3.14159, 0.0, 0.0]), a=A_DEFAULT*ACCEL_FACTOR, v=V_CIRC*SPEED_FACTOR, r=0.002)
  movel(T(p[0.189108, -0.340929, 0.050000, 3.14159, 0.0, 0.0]), a=A_DEFAULT*ACCEL_FACTOR, v=V_CIRC*SPEED_FACTOR, r=0.002)
  movel(T(p[0.191723, -0.334542, 0.050000, 3.14159, 0.0, 0.0]), a=A_DEFAULT*ACCEL_FACTOR, v=V_CIRC*SPEED_FACTOR, r=0.002)
  movel(T(p[0.200047, -0.338511, 0.050000, 3.14159, 0.0, 0.0]), a=A_DEFAULT*ACCEL_FACTOR, v=V_CIRC*SPEED_FACTOR, r=0.002)
  movel(T(p[0.197147, -0.346203, 0.050000, 3.14159, 0.0, 0.0]), a=A_DEFAULT*ACCEL_FACTOR, v=V_CIRC*SPEED_FACTOR, r=0.002)
  movel(T(p[0.192637, -0.342178, 0.050000, 3.14159, 0.0, 0.0]), a=A_DEFAULT*ACCEL_FACTOR, v=V_CIRC*SPEED_FACTOR, r=0.002)
  movel(T(p[0.199941, -0.338712, 0.050000, 3.14159, 0.0, 0.0]), a=A_DEFAULT*ACCEL_FACTOR, v=V_CIRC*SPEED_FACTOR, r=0.002)
  movel(T(p[0.204537, -0.346760, 0.050000, 3.14159, 0.0, 0.0]), a=A_DEFAULT*ACCEL_FACTOR, v=V_CIRC*SPEED_FACTOR, r=0.002)
  movel(T(p[0.198308, -0.350040, 0.050000, 3.14159, 0.0, 0.0]), a=A_DEFAULT*ACCEL_FACTOR, v=V_CIRC*SPEED_FACTOR, r=0.002)
  movel(T(p[0.198743, -0.343549, 0.050000, 3.14159, 0.0, 0.0]), a=A_DEFAULT*ACCEL_FACTOR, v=V_CIRC*SPEED_FACTOR, r=0.002)
  movel(T(p[0.207568, -0.345396, 0.050000, 3.14159, 0.0, 0.0]), a=A_DEFAULT*ACCEL_FACTOR, v=V_CIRC*SPEED_FACTOR, r=0.002)
  movel(T(p[0.206662, -0.353966, 0.050000, 3.14159, 0.0, 0.0]), a=A_DEFAULT*ACCEL_FACTOR, v=V_CIRC*SPEED_FACTOR, r=0.002)
  movel(T(p[0.210965, -0.358063, 0.050000, 3.14159, 0.0, 0.0]), a=A_DEFAULT*ACCEL_FACTOR, v=V_CIRC*SPEED_FACTOR, r=0.002)
  movel(T(p[0.197831, -0.356868, 0.050000, 3.14159, 0.0, 0.0]), a=A_DEFAULT*ACCEL_FACTOR, v=V_CIRC*SPEED_FACTOR, r=0.002)
  movel(T(p[0.197313, -0.354239, 0.050000, 3.14159, 0.0, 0.0]), a=A_DEFAULT*ACCEL_FACTOR, v=V_CIRC*SPEED_FACTOR, r=0.002)
  movel(T(p[0.197882, -0.360567, 0.050000, 3.14159, 0.0, 0.0]), a=A_DEFAULT*ACCEL_FACTOR, v=V_CIRC*SPEED_FACTOR, r=0.002)
  movel(T(p[0.189034, -0.359736, 0.050000, 3.14159, 0.0, 0.0]), a=A_DEFAULT*ACCEL_FACTOR, v=V_CIRC*SPEED_FACTOR, r=0.002)
  movel(T(p[0.188944, -0.350957, 0.050000, 3.14159, 0.0, 0.0]), a=A_DEFAULT*ACCEL_FACTOR, v=V_CIRC*SPEED_FACTOR, r=0.002)
  movel(T(p[0.195069, -0.352240, 0.050000, 3.14159, 0.0, 0.0]), a=A_DEFAULT*ACCEL_FACTOR, v=V_CIRC*SPEED_FACTOR, r=0.002)
  movel(T(p[0.190166, -0.357795, 0.050000, 3.14159, 0.0, 0.0]), a=A_DEFAULT*ACCEL_FACTOR, v=V_CIRC*SPEED_FACTOR, r=0.002)
  movel(T(p[0.183077, -0.351727, 0.050000, 3.14159, 0.0, 0.0]), a=A_DEFAULT*ACCEL_FACTOR, v=V_CIRC*SPEED_FACTOR, r=0.002)
  movel(T(p[0.187816, -0.345635, 0.050000, 3.14159, 0.0, 0.0]), a=A_DEFAULT*ACCEL_FACTOR, v=V_CIRC*SPEED_FACTOR, r=0.002)
  movel(T(p[0.190418, -0.351174, 0.050000, 3.14159, 0.0, 0.0]), a=A_DEFAULT*ACCEL_FACTOR, v=V_CIRC*SPEED_FACTOR, r=0.002)
  movel(T(p[0.181973, -0.352487, 0.050000, 3.14159, 0.0, 0.0]), a=A_DEFAULT*ACCEL_FACTOR, v=V_CIRC*SPEED_FACTOR, r=0.002)
  movel(T(p[0.179702, -0.343713, 0.050000, 3.14159, 0.0, 0.0]), a=A_DEFAULT*ACCEL_FACTOR, v=V_CIRC*SPEED_FACTOR, r=0.002)
  movel(T(p[0.186221, -0.342851, 0.050000, 3.14159, 0.0, 0.0]), a=A_DEFAULT*ACCEL_FACTOR, v=V_CIRC*SPEED_FACTOR, r=0.002)
  movel(T(p[0.183355, -0.349185, 0.050000, 3.14159, 0.0, 0.0]), a=A_DEFAULT*ACCEL_FACTOR, v=V_CIRC*SPEED_FACTOR, r=0.002)
  movel(T(p[0.175128, -0.344978, 0.050000, 3.14159, 0.0, 0.0]), a=A_DEFAULT*ACCEL_FACTOR, v=V_CIRC*SPEED_FACTOR, r=0.002)
  movel(T(p[0.178246, -0.337425, 0.050000, 3.14159, 0.0, 0.0]), a=A_DEFAULT*ACCEL_FACTOR, v=V_CIRC*SPEED_FACTOR, r=0.002)
  movel(T(p[0.182578, -0.341638, 0.050000, 3.14159, 0.0, 0.0]), a=A_DEFAULT*ACCEL_FACTOR, v=V_CIRC*SPEED_FACTOR, r=0.002)
  movel(T(p[0.175123, -0.344896, 0.050000, 3.14159, 0.0, 0.0]), a=A_DEFAULT*ACCEL_FACTOR, v=V_CIRC*SPEED_FACTOR, r=0.002)
  movel(T(p[0.171025, -0.336323, 0.050000, 3.14159, 0.0, 0.0]), a=A_DEFAULT*ACCEL_FACTOR, v=V_CIRC*SPEED_FACTOR, r=0.002)
  movel(T(p[0.177378, -0.333966, 0.050000, 3.14159, 0.0, 0.0]), a=A_DEFAULT*ACCEL_FACTOR, v=V_CIRC*SPEED_FACTOR, r=0.002)
  movel(T(p[0.176172, -0.340413, 0.050000, 3.14159, 0.0, 0.0]), a=A_DEFAULT*ACCEL_FACTOR, v=V_CIRC*SPEED_FACTOR, r=0.002)
  movel(T(p[0.167489, -0.337986, 0.050000, 3.14159, 0.0, 0.0]), a=A_DEFAULT*ACCEL_FACTOR, v=V_CIRC*SPEED_FACTOR, r=0.002)
  end_force_mode()
  movel(T(p[0.168180, -0.338891, 0.060000, 3.14159, 0.0, 0.0]), a=A_DEFAULT*ACCEL_FACTOR, v=V_APPROACH*SPEED_FACTOR)
end

def cycle_4():
  # --- Cycle 4 - Rectiligne (0deg) ---
  movel(T(p[0.200000, -0.305657, 0.060000, 3.14159, 0.0, 0.0]), a=A_DEFAULT*ACCEL_FACTOR, v=V_APPROACH*SPEED_FACTOR)
  movel(T(p[0.200000, -0.305657, 0.050000, 3.14159, 0.0, 0.0]), a=A_DEFAULT*ACCEL_FACTOR, v=V_CONTACT*SPEED_FACTOR)
  force_mode(get_actual_tcp_pose(), [0, 0, 1, 0, 0, 0], [0, 0, -6.0, 0, 0, 0], 2, [0.002, 0.002, 0.04, 0.35, 0.35, 0.35])
  movel(T(p[0.195151, -0.310505, 0.050000, 3.14159, 0.0, 0.0]), a=A_DEFAULT*ACCEL_FACTOR, v=V_RECT*SPEED_FACTOR, r=0.002)
  movel(T(p[0.190303, -0.315354, 0.050000, 3.14159, 0.0, 0.0]), a=A_DEFAULT*ACCEL_FACTOR, v=V_RECT*SPEED_FACTOR, r=0.002)
  movel(T(p[0.185454, -0.320203, 0.050000, 3.14159, 0.0, 0.0]), a=A_DEFAULT*ACCEL_FACTOR, v=V_RECT*SPEED_FACTOR, r=0.002)
  movel(T(p[0.180605, -0.325052, 0.050000, 3.14159, 0.0, 0.0]), a=A_DEFAULT*ACCEL_FACTOR, v=V_RECT*SPEED_FACTOR, r=0.002)
  movel(T(p[0.175756, -0.329901, 0.050000, 3.14159, 0.0, 0.0]), a=A_DEFAULT*ACCEL_FACTOR, v=V_RECT*SPEED_FACTOR, r=0.002)
  movel(T(p[0.170908, -0.334749, 0.050000, 3.14159, 0.0, 0.0]), a=A_DEFAULT*ACCEL_FACTOR, v=V_RECT*SPEED_FACTOR, r=0.002)
  movel(T(p[0.176413, -0.334194, 0.050000, 3.14159, 0.0, 0.0]), a=A_DEFAULT*ACCEL_FACTOR, v=V_RECT*SPEED_FACTOR, r=0.002)
  movel(T(p[0.181262, -0.329345, 0.050000, 3.14159, 0.0, 0.0]), a=A_DEFAULT*ACCEL_FACTOR, v=V_RECT*SPEED_FACTOR, r=0.002)
  movel(T(p[0.186110, -0.324496, 0.050000, 3.14159, 0.0, 0.0]), a=A_DEFAULT*ACCEL_FACTOR, v=V_RECT*SPEED_FACTOR, r=0.002)
  movel(T(p[0.190959, -0.319648, 0.050000, 3.14159, 0.0, 0.0]), a=A_DEFAULT*ACCEL_FACTOR, v=V_RECT*SPEED_FACTOR, r=0.002)
  movel(T(p[0.195808, -0.314799, 0.050000, 3.14159, 0.0, 0.0]), a=A_DEFAULT*ACCEL_FACTOR, v=V_RECT*SPEED_FACTOR, r=0.002)
  movel(T(p[0.200657, -0.309950, 0.050000, 3.14159, 0.0, 0.0]), a=A_DEFAULT*ACCEL_FACTOR, v=V_RECT*SPEED_FACTOR, r=0.002)
  movel(T(p[0.202525, -0.313031, 0.050000, 3.14159, 0.0, 0.0]), a=A_DEFAULT*ACCEL_FACTOR, v=V_RECT*SPEED_FACTOR, r=0.002)
  movel(T(p[0.197676, -0.317880, 0.050000, 3.14159, 0.0, 0.0]), a=A_DEFAULT*ACCEL_FACTOR, v=V_RECT*SPEED_FACTOR, r=0.002)
  movel(T(p[0.192828, -0.322729, 0.050000, 3.14159, 0.0, 0.0]), a=A_DEFAULT*ACCEL_FACTOR, v=V_RECT*SPEED_FACTOR, r=0.002)
  movel(T(p[0.187979, -0.327577, 0.050000, 3.14159, 0.0, 0.0]), a=A_DEFAULT*ACCEL_FACTOR, v=V_RECT*SPEED_FACTOR, r=0.002)
  movel(T(p[0.183131, -0.332426, 0.050000, 3.14159, 0.0, 0.0]), a=A_DEFAULT*ACCEL_FACTOR, v=V_RECT*SPEED_FACTOR, r=0.002)
  movel(T(p[0.178282, -0.337274, 0.050000, 3.14159, 0.0, 0.0]), a=A_DEFAULT*ACCEL_FACTOR, v=V_RECT*SPEED_FACTOR, r=0.002)
  movel(T(p[0.178938, -0.341568, 0.050000, 3.14159, 0.0, 0.0]), a=A_DEFAULT*ACCEL_FACTOR, v=V_RECT*SPEED_FACTOR, r=0.002)
  movel(T(p[0.183787, -0.336719, 0.050000, 3.14159, 0.0, 0.0]), a=A_DEFAULT*ACCEL_FACTOR, v=V_RECT*SPEED_FACTOR, r=0.002)
  movel(T(p[0.188636, -0.331870, 0.050000, 3.14159, 0.0, 0.0]), a=A_DEFAULT*ACCEL_FACTOR, v=V_RECT*SPEED_FACTOR, r=0.002)
  movel(T(p[0.193485, -0.327021, 0.050000, 3.14159, 0.0, 0.0]), a=A_DEFAULT*ACCEL_FACTOR, v=V_RECT*SPEED_FACTOR, r=0.002)
  movel(T(p[0.198333, -0.322173, 0.050000, 3.14159, 0.0, 0.0]), a=A_DEFAULT*ACCEL_FACTOR, v=V_RECT*SPEED_FACTOR, r=0.002)
  movel(T(p[0.203182, -0.317324, 0.050000, 3.14159, 0.0, 0.0]), a=A_DEFAULT*ACCEL_FACTOR, v=V_RECT*SPEED_FACTOR, r=0.002)
  movel(T(p[0.209899, -0.315556, 0.050000, 3.14159, 0.0, 0.0]), a=A_DEFAULT*ACCEL_FACTOR, v=V_RECT*SPEED_FACTOR, r=0.002)
  movel(T(p[0.205051, -0.320405, 0.050000, 3.14159, 0.0, 0.0]), a=A_DEFAULT*ACCEL_FACTOR, v=V_RECT*SPEED_FACTOR, r=0.002)
  movel(T(p[0.200202, -0.325254, 0.050000, 3.14159, 0.0, 0.0]), a=A_DEFAULT*ACCEL_FACTOR, v=V_RECT*SPEED_FACTOR, r=0.002)
  movel(T(p[0.195354, -0.330102, 0.050000, 3.14159, 0.0, 0.0]), a=A_DEFAULT*ACCEL_FACTOR, v=V_RECT*SPEED_FACTOR, r=0.002)
  movel(T(p[0.190504, -0.334952, 0.050000, 3.14159, 0.0, 0.0]), a=A_DEFAULT*ACCEL_FACTOR, v=V_RECT*SPEED_FACTOR, r=0.002)
  movel(T(p[0.185656, -0.339800, 0.050000, 3.14159, 0.0, 0.0]), a=A_DEFAULT*ACCEL_FACTOR, v=V_RECT*SPEED_FACTOR, r=0.002)
  movel(T(p[0.180807, -0.344649, 0.050000, 3.14159, 0.0, 0.0]), a=A_DEFAULT*ACCEL_FACTOR, v=V_RECT*SPEED_FACTOR, r=0.002)
  movel(T(p[0.186313, -0.344093, 0.050000, 3.14159, 0.0, 0.0]), a=A_DEFAULT*ACCEL_FACTOR, v=V_RECT*SPEED_FACTOR, r=0.002)
  movel(T(p[0.191161, -0.339244, 0.050000, 3.14159, 0.0, 0.0]), a=A_DEFAULT*ACCEL_FACTOR, v=V_RECT*SPEED_FACTOR, r=0.002)
  movel(T(p[0.196010, -0.334396, 0.050000, 3.14159, 0.0, 0.0]), a=A_DEFAULT*ACCEL_FACTOR, v=V_RECT*SPEED_FACTOR, r=0.002)
  movel(T(p[0.200858, -0.329547, 0.050000, 3.14159, 0.0, 0.0]), a=A_DEFAULT*ACCEL_FACTOR, v=V_RECT*SPEED_FACTOR, r=0.002)
  movel(T(p[0.205707, -0.324699, 0.050000, 3.14159, 0.0, 0.0]), a=A_DEFAULT*ACCEL_FACTOR, v=V_RECT*SPEED_FACTOR, r=0.002)
  movel(T(p[0.210556, -0.319849, 0.050000, 3.14159, 0.0, 0.0]), a=A_DEFAULT*ACCEL_FACTOR, v=V_RECT*SPEED_FACTOR, r=0.002)
  movel(T(p[0.212425, -0.322931, 0.050000, 3.14159, 0.0, 0.0]), a=A_DEFAULT*ACCEL_FACTOR, v=V_RECT*SPEED_FACTOR, r=0.002)
  movel(T(p[0.207576, -0.327779, 0.050000, 3.14159, 0.0, 0.0]), a=A_DEFAULT*ACCEL_FACTOR, v=V_RECT*SPEED_FACTOR, r=0.002)
  movel(T(p[0.202727, -0.332628, 0.050000, 3.14159, 0.0, 0.0]), a=A_DEFAULT*ACCEL_FACTOR, v=V_RECT*SPEED_FACTOR, r=0.002)
  movel(T(p[0.197879, -0.337477, 0.050000, 3.14159, 0.0, 0.0]), a=A_DEFAULT*ACCEL_FACTOR, v=V_RECT*SPEED_FACTOR, r=0.002)
  movel(T(p[0.193030, -0.342325, 0.050000, 3.14159, 0.0, 0.0]), a=A_DEFAULT*ACCEL_FACTOR, v=V_RECT*SPEED_FACTOR, r=0.002)
  movel(T(p[0.188181, -0.347174, 0.050000, 3.14159, 0.0, 0.0]), a=A_DEFAULT*ACCEL_FACTOR, v=V_RECT*SPEED_FACTOR, r=0.002)
  movel(T(p[0.188838, -0.351467, 0.050000, 3.14159, 0.0, 0.0]), a=A_DEFAULT*ACCEL_FACTOR, v=V_RECT*SPEED_FACTOR, r=0.002)
  movel(T(p[0.193686, -0.346619, 0.050000, 3.14159, 0.0, 0.0]), a=A_DEFAULT*ACCEL_FACTOR, v=V_RECT*SPEED_FACTOR, r=0.002)
  movel(T(p[0.198536, -0.341770, 0.050000, 3.14159, 0.0, 0.0]), a=A_DEFAULT*ACCEL_FACTOR, v=V_RECT*SPEED_FACTOR, r=0.002)
  movel(T(p[0.203384, -0.336921, 0.050000, 3.14159, 0.0, 0.0]), a=A_DEFAULT*ACCEL_FACTOR, v=V_RECT*SPEED_FACTOR, r=0.002)
  movel(T(p[0.208233, -0.332072, 0.050000, 3.14159, 0.0, 0.0]), a=A_DEFAULT*ACCEL_FACTOR, v=V_RECT*SPEED_FACTOR, r=0.002)
  movel(T(p[0.213081, -0.327224, 0.050000, 3.14159, 0.0, 0.0]), a=A_DEFAULT*ACCEL_FACTOR, v=V_RECT*SPEED_FACTOR, r=0.002)
  movel(T(p[0.219799, -0.325456, 0.050000, 3.14159, 0.0, 0.0]), a=A_DEFAULT*ACCEL_FACTOR, v=V_RECT*SPEED_FACTOR, r=0.002)
  movel(T(p[0.214950, -0.330304, 0.050000, 3.14159, 0.0, 0.0]), a=A_DEFAULT*ACCEL_FACTOR, v=V_RECT*SPEED_FACTOR, r=0.002)
  movel(T(p[0.210102, -0.335153, 0.050000, 3.14159, 0.0, 0.0]), a=A_DEFAULT*ACCEL_FACTOR, v=V_RECT*SPEED_FACTOR, r=0.002)
  movel(T(p[0.205253, -0.340002, 0.050000, 3.14159, 0.0, 0.0]), a=A_DEFAULT*ACCEL_FACTOR, v=V_RECT*SPEED_FACTOR, r=0.002)
  movel(T(p[0.200404, -0.344851, 0.050000, 3.14159, 0.0, 0.0]), a=A_DEFAULT*ACCEL_FACTOR, v=V_RECT*SPEED_FACTOR, r=0.002)
  movel(T(p[0.195555, -0.349700, 0.050000, 3.14159, 0.0, 0.0]), a=A_DEFAULT*ACCEL_FACTOR, v=V_RECT*SPEED_FACTOR, r=0.002)
  movel(T(p[0.190706, -0.354548, 0.050000, 3.14159, 0.0, 0.0]), a=A_DEFAULT*ACCEL_FACTOR, v=V_RECT*SPEED_FACTOR, r=0.002)
  movel(T(p[0.196212, -0.353993, 0.050000, 3.14159, 0.0, 0.0]), a=A_DEFAULT*ACCEL_FACTOR, v=V_RECT*SPEED_FACTOR, r=0.002)
  movel(T(p[0.201061, -0.349144, 0.050000, 3.14159, 0.0, 0.0]), a=A_DEFAULT*ACCEL_FACTOR, v=V_RECT*SPEED_FACTOR, r=0.002)
  movel(T(p[0.205909, -0.344295, 0.050000, 3.14159, 0.0, 0.0]), a=A_DEFAULT*ACCEL_FACTOR, v=V_RECT*SPEED_FACTOR, r=0.002)
  movel(T(p[0.210758, -0.339447, 0.050000, 3.14159, 0.0, 0.0]), a=A_DEFAULT*ACCEL_FACTOR, v=V_RECT*SPEED_FACTOR, r=0.002)
  movel(T(p[0.215607, -0.334598, 0.050000, 3.14159, 0.0, 0.0]), a=A_DEFAULT*ACCEL_FACTOR, v=V_RECT*SPEED_FACTOR, r=0.002)
  movel(T(p[0.220456, -0.329749, 0.050000, 3.14159, 0.0, 0.0]), a=A_DEFAULT*ACCEL_FACTOR, v=V_RECT*SPEED_FACTOR, r=0.002)
  movel(T(p[0.222324, -0.332830, 0.050000, 3.14159, 0.0, 0.0]), a=A_DEFAULT*ACCEL_FACTOR, v=V_RECT*SPEED_FACTOR, r=0.002)
  movel(T(p[0.217475, -0.337679, 0.050000, 3.14159, 0.0, 0.0]), a=A_DEFAULT*ACCEL_FACTOR, v=V_RECT*SPEED_FACTOR, r=0.002)
  movel(T(p[0.212627, -0.342528, 0.050000, 3.14159, 0.0, 0.0]), a=A_DEFAULT*ACCEL_FACTOR, v=V_RECT*SPEED_FACTOR, r=0.002)
  movel(T(p[0.207778, -0.347376, 0.050000, 3.14159, 0.0, 0.0]), a=A_DEFAULT*ACCEL_FACTOR, v=V_RECT*SPEED_FACTOR, r=0.002)
  movel(T(p[0.202930, -0.352225, 0.050000, 3.14159, 0.0, 0.0]), a=A_DEFAULT*ACCEL_FACTOR, v=V_RECT*SPEED_FACTOR, r=0.002)
  movel(T(p[0.198081, -0.357073, 0.050000, 3.14159, 0.0, 0.0]), a=A_DEFAULT*ACCEL_FACTOR, v=V_RECT*SPEED_FACTOR, r=0.002)
  movel(T(p[0.198737, -0.361367, 0.050000, 3.14159, 0.0, 0.0]), a=A_DEFAULT*ACCEL_FACTOR, v=V_RECT*SPEED_FACTOR, r=0.002)
  movel(T(p[0.203586, -0.356518, 0.050000, 3.14159, 0.0, 0.0]), a=A_DEFAULT*ACCEL_FACTOR, v=V_RECT*SPEED_FACTOR, r=0.002)
  movel(T(p[0.208435, -0.351669, 0.050000, 3.14159, 0.0, 0.0]), a=A_DEFAULT*ACCEL_FACTOR, v=V_RECT*SPEED_FACTOR, r=0.002)
  movel(T(p[0.213284, -0.346820, 0.050000, 3.14159, 0.0, 0.0]), a=A_DEFAULT*ACCEL_FACTOR, v=V_RECT*SPEED_FACTOR, r=0.002)
  movel(T(p[0.218132, -0.341972, 0.050000, 3.14159, 0.0, 0.0]), a=A_DEFAULT*ACCEL_FACTOR, v=V_RECT*SPEED_FACTOR, r=0.002)
  movel(T(p[0.222981, -0.337123, 0.050000, 3.14159, 0.0, 0.0]), a=A_DEFAULT*ACCEL_FACTOR, v=V_RECT*SPEED_FACTOR, r=0.002)
  movel(T(p[0.229698, -0.335355, 0.050000, 3.14159, 0.0, 0.0]), a=A_DEFAULT*ACCEL_FACTOR, v=V_RECT*SPEED_FACTOR, r=0.002)
  movel(T(p[0.224850, -0.340204, 0.050000, 3.14159, 0.0, 0.0]), a=A_DEFAULT*ACCEL_FACTOR, v=V_RECT*SPEED_FACTOR, r=0.002)
  movel(T(p[0.220001, -0.345053, 0.050000, 3.14159, 0.0, 0.0]), a=A_DEFAULT*ACCEL_FACTOR, v=V_RECT*SPEED_FACTOR, r=0.002)
  movel(T(p[0.215153, -0.349901, 0.050000, 3.14159, 0.0, 0.0]), a=A_DEFAULT*ACCEL_FACTOR, v=V_RECT*SPEED_FACTOR, r=0.002)
  movel(T(p[0.210303, -0.354751, 0.050000, 3.14159, 0.0, 0.0]), a=A_DEFAULT*ACCEL_FACTOR, v=V_RECT*SPEED_FACTOR, r=0.002)
  movel(T(p[0.205455, -0.359599, 0.050000, 3.14159, 0.0, 0.0]), a=A_DEFAULT*ACCEL_FACTOR, v=V_RECT*SPEED_FACTOR, r=0.002)
  movel(T(p[0.200606, -0.364448, 0.050000, 3.14159, 0.0, 0.0]), a=A_DEFAULT*ACCEL_FACTOR, v=V_RECT*SPEED_FACTOR, r=0.002)
  end_force_mode()
  movel(T(p[0.200000, -0.365054, 0.060000, 3.14159, 0.0, 0.0]), a=A_DEFAULT*ACCEL_FACTOR, v=V_APPROACH*SPEED_FACTOR)
end

def cycle_5():
  # --- Cycle 5 - Rectiligne (90deg) ---
  movel(T(p[0.170302, -0.335355, 0.060000, 3.14159, 0.0, 0.0]), a=A_DEFAULT*ACCEL_FACTOR, v=V_APPROACH*SPEED_FACTOR)
  movel(T(p[0.170302, -0.335355, 0.050000, 3.14159, 0.0, 0.0]), a=A_DEFAULT*ACCEL_FACTOR, v=V_CONTACT*SPEED_FACTOR)
  force_mode(get_actual_tcp_pose(), [0, 0, 1, 0, 0, 0], [0, 0, -6.0, 0, 0, 0], 2, [0.002, 0.002, 0.04, 0.35, 0.35, 0.35])
  movel(T(p[0.175150, -0.340204, 0.050000, 3.14159, 0.0, 0.0]), a=A_DEFAULT*ACCEL_FACTOR, v=V_RECT*SPEED_FACTOR, r=0.002)
  movel(T(p[0.179999, -0.345053, 0.050000, 3.14159, 0.0, 0.0]), a=A_DEFAULT*ACCEL_FACTOR, v=V_RECT*SPEED_FACTOR, r=0.002)
  movel(T(p[0.184847, -0.349901, 0.050000, 3.14159, 0.0, 0.0]), a=A_DEFAULT*ACCEL_FACTOR, v=V_RECT*SPEED_FACTOR, r=0.002)
  movel(T(p[0.189697, -0.354751, 0.050000, 3.14159, 0.0, 0.0]), a=A_DEFAULT*ACCEL_FACTOR, v=V_RECT*SPEED_FACTOR, r=0.002)
  movel(T(p[0.194545, -0.359599, 0.050000, 3.14159, 0.0, 0.0]), a=A_DEFAULT*ACCEL_FACTOR, v=V_RECT*SPEED_FACTOR, r=0.002)
  movel(T(p[0.199394, -0.364448, 0.050000, 3.14159, 0.0, 0.0]), a=A_DEFAULT*ACCEL_FACTOR, v=V_RECT*SPEED_FACTOR, r=0.002)
  movel(T(p[0.198838, -0.358942, 0.050000, 3.14159, 0.0, 0.0]), a=A_DEFAULT*ACCEL_FACTOR, v=V_RECT*SPEED_FACTOR, r=0.002)
  movel(T(p[0.193990, -0.354094, 0.050000, 3.14159, 0.0, 0.0]), a=A_DEFAULT*ACCEL_FACTOR, v=V_RECT*SPEED_FACTOR, r=0.002)
  movel(T(p[0.189141, -0.349245, 0.050000, 3.14159, 0.0, 0.0]), a=A_DEFAULT*ACCEL_FACTOR, v=V_RECT*SPEED_FACTOR, r=0.002)
  movel(T(p[0.184292, -0.344396, 0.050000, 3.14159, 0.0, 0.0]), a=A_DEFAULT*ACCEL_FACTOR, v=V_RECT*SPEED_FACTOR, r=0.002)
  movel(T(p[0.179444, -0.339548, 0.050000, 3.14159, 0.0, 0.0]), a=A_DEFAULT*ACCEL_FACTOR, v=V_RECT*SPEED_FACTOR, r=0.002)
  movel(T(p[0.174594, -0.334698, 0.050000, 3.14159, 0.0, 0.0]), a=A_DEFAULT*ACCEL_FACTOR, v=V_RECT*SPEED_FACTOR, r=0.002)
  movel(T(p[0.177676, -0.332830, 0.050000, 3.14159, 0.0, 0.0]), a=A_DEFAULT*ACCEL_FACTOR, v=V_RECT*SPEED_FACTOR, r=0.002)
  movel(T(p[0.182525, -0.337679, 0.050000, 3.14159, 0.0, 0.0]), a=A_DEFAULT*ACCEL_FACTOR, v=V_RECT*SPEED_FACTOR, r=0.002)
  movel(T(p[0.187373, -0.342528, 0.050000, 3.14159, 0.0, 0.0]), a=A_DEFAULT*ACCEL_FACTOR, v=V_RECT*SPEED_FACTOR, r=0.002)
  movel(T(p[0.192222, -0.347376, 0.050000, 3.14159, 0.0, 0.0]), a=A_DEFAULT*ACCEL_FACTOR, v=V_RECT*SPEED_FACTOR, r=0.002)
  movel(T(p[0.197070, -0.352225, 0.050000, 3.14159, 0.0, 0.0]), a=A_DEFAULT*ACCEL_FACTOR, v=V_RECT*SPEED_FACTOR, r=0.002)
  movel(T(p[0.201919, -0.357073, 0.050000, 3.14159, 0.0, 0.0]), a=A_DEFAULT*ACCEL_FACTOR, v=V_RECT*SPEED_FACTOR, r=0.002)
  movel(T(p[0.206213, -0.356417, 0.050000, 3.14159, 0.0, 0.0]), a=A_DEFAULT*ACCEL_FACTOR, v=V_RECT*SPEED_FACTOR, r=0.002)
  movel(T(p[0.201364, -0.351569, 0.050000, 3.14159, 0.0, 0.0]), a=A_DEFAULT*ACCEL_FACTOR, v=V_RECT*SPEED_FACTOR, r=0.002)
  movel(T(p[0.196515, -0.346719, 0.050000, 3.14159, 0.0, 0.0]), a=A_DEFAULT*ACCEL_FACTOR, v=V_RECT*SPEED_FACTOR, r=0.002)
  movel(T(p[0.191666, -0.341871, 0.050000, 3.14159, 0.0, 0.0]), a=A_DEFAULT*ACCEL_FACTOR, v=V_RECT*SPEED_FACTOR, r=0.002)
  movel(T(p[0.186817, -0.337022, 0.050000, 3.14159, 0.0, 0.0]), a=A_DEFAULT*ACCEL_FACTOR, v=V_RECT*SPEED_FACTOR, r=0.002)
  movel(T(p[0.181969, -0.332173, 0.050000, 3.14159, 0.0, 0.0]), a=A_DEFAULT*ACCEL_FACTOR, v=V_RECT*SPEED_FACTOR, r=0.002)
  movel(T(p[0.180201, -0.325456, 0.050000, 3.14159, 0.0, 0.0]), a=A_DEFAULT*ACCEL_FACTOR, v=V_RECT*SPEED_FACTOR, r=0.002)
  movel(T(p[0.185050, -0.330304, 0.050000, 3.14159, 0.0, 0.0]), a=A_DEFAULT*ACCEL_FACTOR, v=V_RECT*SPEED_FACTOR, r=0.002)
  movel(T(p[0.189898, -0.335153, 0.050000, 3.14159, 0.0, 0.0]), a=A_DEFAULT*ACCEL_FACTOR, v=V_RECT*SPEED_FACTOR, r=0.002)
  movel(T(p[0.194747, -0.340002, 0.050000, 3.14159, 0.0, 0.0]), a=A_DEFAULT*ACCEL_FACTOR, v=V_RECT*SPEED_FACTOR, r=0.002)
  movel(T(p[0.199596, -0.344851, 0.050000, 3.14159, 0.0, 0.0]), a=A_DEFAULT*ACCEL_FACTOR, v=V_RECT*SPEED_FACTOR, r=0.002)
  movel(T(p[0.204445, -0.349700, 0.050000, 3.14159, 0.0, 0.0]), a=A_DEFAULT*ACCEL_FACTOR, v=V_RECT*SPEED_FACTOR, r=0.002)
  movel(T(p[0.209294, -0.354548, 0.050000, 3.14159, 0.0, 0.0]), a=A_DEFAULT*ACCEL_FACTOR, v=V_RECT*SPEED_FACTOR, r=0.002)
  movel(T(p[0.208738, -0.349043, 0.050000, 3.14159, 0.0, 0.0]), a=A_DEFAULT*ACCEL_FACTOR, v=V_RECT*SPEED_FACTOR, r=0.002)
  movel(T(p[0.203889, -0.344194, 0.050000, 3.14159, 0.0, 0.0]), a=A_DEFAULT*ACCEL_FACTOR, v=V_RECT*SPEED_FACTOR, r=0.002)
  movel(T(p[0.199040, -0.339346, 0.050000, 3.14159, 0.0, 0.0]), a=A_DEFAULT*ACCEL_FACTOR, v=V_RECT*SPEED_FACTOR, r=0.002)
  movel(T(p[0.194192, -0.334497, 0.050000, 3.14159, 0.0, 0.0]), a=A_DEFAULT*ACCEL_FACTOR, v=V_RECT*SPEED_FACTOR, r=0.002)
  movel(T(p[0.189343, -0.329648, 0.050000, 3.14159, 0.0, 0.0]), a=A_DEFAULT*ACCEL_FACTOR, v=V_RECT*SPEED_FACTOR, r=0.002)
  movel(T(p[0.184494, -0.324799, 0.050000, 3.14159, 0.0, 0.0]), a=A_DEFAULT*ACCEL_FACTOR, v=V_RECT*SPEED_FACTOR, r=0.002)
  movel(T(p[0.187575, -0.322931, 0.050000, 3.14159, 0.0, 0.0]), a=A_DEFAULT*ACCEL_FACTOR, v=V_RECT*SPEED_FACTOR, r=0.002)
  movel(T(p[0.192424, -0.327779, 0.050000, 3.14159, 0.0, 0.0]), a=A_DEFAULT*ACCEL_FACTOR, v=V_RECT*SPEED_FACTOR, r=0.002)
  movel(T(p[0.197273, -0.332628, 0.050000, 3.14159, 0.0, 0.0]), a=A_DEFAULT*ACCEL_FACTOR, v=V_RECT*SPEED_FACTOR, r=0.002)
  movel(T(p[0.202121, -0.337477, 0.050000, 3.14159, 0.0, 0.0]), a=A_DEFAULT*ACCEL_FACTOR, v=V_RECT*SPEED_FACTOR, r=0.002)
  movel(T(p[0.206970, -0.342325, 0.050000, 3.14159, 0.0, 0.0]), a=A_DEFAULT*ACCEL_FACTOR, v=V_RECT*SPEED_FACTOR, r=0.002)
  movel(T(p[0.211819, -0.347174, 0.050000, 3.14159, 0.0, 0.0]), a=A_DEFAULT*ACCEL_FACTOR, v=V_RECT*SPEED_FACTOR, r=0.002)
  movel(T(p[0.216112, -0.346518, 0.050000, 3.14159, 0.0, 0.0]), a=A_DEFAULT*ACCEL_FACTOR, v=V_RECT*SPEED_FACTOR, r=0.002)
  movel(T(p[0.211264, -0.341669, 0.050000, 3.14159, 0.0, 0.0]), a=A_DEFAULT*ACCEL_FACTOR, v=V_RECT*SPEED_FACTOR, r=0.002)
  movel(T(p[0.206414, -0.336820, 0.050000, 3.14159, 0.0, 0.0]), a=A_DEFAULT*ACCEL_FACTOR, v=V_RECT*SPEED_FACTOR, r=0.002)
  movel(T(p[0.201566, -0.331971, 0.050000, 3.14159, 0.0, 0.0]), a=A_DEFAULT*ACCEL_FACTOR, v=V_RECT*SPEED_FACTOR, r=0.002)
  movel(T(p[0.196717, -0.327122, 0.050000, 3.14159, 0.0, 0.0]), a=A_DEFAULT*ACCEL_FACTOR, v=V_RECT*SPEED_FACTOR, r=0.002)
  movel(T(p[0.191868, -0.322274, 0.050000, 3.14159, 0.0, 0.0]), a=A_DEFAULT*ACCEL_FACTOR, v=V_RECT*SPEED_FACTOR, r=0.002)
  movel(T(p[0.190101, -0.315556, 0.050000, 3.14159, 0.0, 0.0]), a=A_DEFAULT*ACCEL_FACTOR, v=V_RECT*SPEED_FACTOR, r=0.002)
  movel(T(p[0.194949, -0.320405, 0.050000, 3.14159, 0.0, 0.0]), a=A_DEFAULT*ACCEL_FACTOR, v=V_RECT*SPEED_FACTOR, r=0.002)
  movel(T(p[0.199798, -0.325254, 0.050000, 3.14159, 0.0, 0.0]), a=A_DEFAULT*ACCEL_FACTOR, v=V_RECT*SPEED_FACTOR, r=0.002)
  movel(T(p[0.204646, -0.330102, 0.050000, 3.14159, 0.0, 0.0]), a=A_DEFAULT*ACCEL_FACTOR, v=V_RECT*SPEED_FACTOR, r=0.002)
  movel(T(p[0.209496, -0.334952, 0.050000, 3.14159, 0.0, 0.0]), a=A_DEFAULT*ACCEL_FACTOR, v=V_RECT*SPEED_FACTOR, r=0.002)
  movel(T(p[0.214344, -0.339800, 0.050000, 3.14159, 0.0, 0.0]), a=A_DEFAULT*ACCEL_FACTOR, v=V_RECT*SPEED_FACTOR, r=0.002)
  movel(T(p[0.219193, -0.344649, 0.050000, 3.14159, 0.0, 0.0]), a=A_DEFAULT*ACCEL_FACTOR, v=V_RECT*SPEED_FACTOR, r=0.002)
  movel(T(p[0.218637, -0.339143, 0.050000, 3.14159, 0.0, 0.0]), a=A_DEFAULT*ACCEL_FACTOR, v=V_RECT*SPEED_FACTOR, r=0.002)
  movel(T(p[0.213789, -0.334295, 0.050000, 3.14159, 0.0, 0.0]), a=A_DEFAULT*ACCEL_FACTOR, v=V_RECT*SPEED_FACTOR, r=0.002)
  movel(T(p[0.208940, -0.329446, 0.050000, 3.14159, 0.0, 0.0]), a=A_DEFAULT*ACCEL_FACTOR, v=V_RECT*SPEED_FACTOR, r=0.002)
  movel(T(p[0.204091, -0.324597, 0.050000, 3.14159, 0.0, 0.0]), a=A_DEFAULT*ACCEL_FACTOR, v=V_RECT*SPEED_FACTOR, r=0.002)
  movel(T(p[0.199243, -0.319749, 0.050000, 3.14159, 0.0, 0.0]), a=A_DEFAULT*ACCEL_FACTOR, v=V_RECT*SPEED_FACTOR, r=0.002)
  movel(T(p[0.194393, -0.314899, 0.050000, 3.14159, 0.0, 0.0]), a=A_DEFAULT*ACCEL_FACTOR, v=V_RECT*SPEED_FACTOR, r=0.002)
  movel(T(p[0.197475, -0.313031, 0.050000, 3.14159, 0.0, 0.0]), a=A_DEFAULT*ACCEL_FACTOR, v=V_RECT*SPEED_FACTOR, r=0.002)
  movel(T(p[0.202324, -0.317880, 0.050000, 3.14159, 0.0, 0.0]), a=A_DEFAULT*ACCEL_FACTOR, v=V_RECT*SPEED_FACTOR, r=0.002)
  movel(T(p[0.207172, -0.322729, 0.050000, 3.14159, 0.0, 0.0]), a=A_DEFAULT*ACCEL_FACTOR, v=V_RECT*SPEED_FACTOR, r=0.002)
  movel(T(p[0.212021, -0.327577, 0.050000, 3.14159, 0.0, 0.0]), a=A_DEFAULT*ACCEL_FACTOR, v=V_RECT*SPEED_FACTOR, r=0.002)
  movel(T(p[0.216869, -0.332426, 0.050000, 3.14159, 0.0, 0.0]), a=A_DEFAULT*ACCEL_FACTOR, v=V_RECT*SPEED_FACTOR, r=0.002)
  movel(T(p[0.221718, -0.337274, 0.050000, 3.14159, 0.0, 0.0]), a=A_DEFAULT*ACCEL_FACTOR, v=V_RECT*SPEED_FACTOR, r=0.002)
  movel(T(p[0.226012, -0.336618, 0.050000, 3.14159, 0.0, 0.0]), a=A_DEFAULT*ACCEL_FACTOR, v=V_RECT*SPEED_FACTOR, r=0.002)
  movel(T(p[0.221163, -0.331770, 0.050000, 3.14159, 0.0, 0.0]), a=A_DEFAULT*ACCEL_FACTOR, v=V_RECT*SPEED_FACTOR, r=0.002)
  movel(T(p[0.216314, -0.326920, 0.050000, 3.14159, 0.0, 0.0]), a=A_DEFAULT*ACCEL_FACTOR, v=V_RECT*SPEED_FACTOR, r=0.002)
  movel(T(p[0.211465, -0.322072, 0.050000, 3.14159, 0.0, 0.0]), a=A_DEFAULT*ACCEL_FACTOR, v=V_RECT*SPEED_FACTOR, r=0.002)
  movel(T(p[0.206616, -0.317223, 0.050000, 3.14159, 0.0, 0.0]), a=A_DEFAULT*ACCEL_FACTOR, v=V_RECT*SPEED_FACTOR, r=0.002)
  movel(T(p[0.201768, -0.312374, 0.050000, 3.14159, 0.0, 0.0]), a=A_DEFAULT*ACCEL_FACTOR, v=V_RECT*SPEED_FACTOR, r=0.002)
  movel(T(p[0.200000, -0.305657, 0.050000, 3.14159, 0.0, 0.0]), a=A_DEFAULT*ACCEL_FACTOR, v=V_RECT*SPEED_FACTOR, r=0.002)
  movel(T(p[0.204849, -0.310505, 0.050000, 3.14159, 0.0, 0.0]), a=A_DEFAULT*ACCEL_FACTOR, v=V_RECT*SPEED_FACTOR, r=0.002)
  movel(T(p[0.209697, -0.315354, 0.050000, 3.14159, 0.0, 0.0]), a=A_DEFAULT*ACCEL_FACTOR, v=V_RECT*SPEED_FACTOR, r=0.002)
  movel(T(p[0.214546, -0.320203, 0.050000, 3.14159, 0.0, 0.0]), a=A_DEFAULT*ACCEL_FACTOR, v=V_RECT*SPEED_FACTOR, r=0.002)
  movel(T(p[0.219395, -0.325052, 0.050000, 3.14159, 0.0, 0.0]), a=A_DEFAULT*ACCEL_FACTOR, v=V_RECT*SPEED_FACTOR, r=0.002)
  movel(T(p[0.224244, -0.329901, 0.050000, 3.14159, 0.0, 0.0]), a=A_DEFAULT*ACCEL_FACTOR, v=V_RECT*SPEED_FACTOR, r=0.002)
  movel(T(p[0.229092, -0.334749, 0.050000, 3.14159, 0.0, 0.0]), a=A_DEFAULT*ACCEL_FACTOR, v=V_RECT*SPEED_FACTOR, r=0.002)
  end_force_mode()
  movel(T(p[0.229698, -0.335355, 0.060000, 3.14159, 0.0, 0.0]), a=A_DEFAULT*ACCEL_FACTOR, v=V_APPROACH*SPEED_FACTOR)
end

def cycle_6():
  # --- Cycle 6 - Rectiligne (0deg) ---
  movel(T(p[0.200000, -0.305657, 0.060000, 3.14159, 0.0, 0.0]), a=A_DEFAULT*ACCEL_FACTOR, v=V_APPROACH*SPEED_FACTOR)
  movel(T(p[0.200000, -0.305657, 0.050000, 3.14159, 0.0, 0.0]), a=A_DEFAULT*ACCEL_FACTOR, v=V_CONTACT*SPEED_FACTOR)
  force_mode(get_actual_tcp_pose(), [0, 0, 1, 0, 0, 0], [0, 0, -6.0, 0, 0, 0], 2, [0.002, 0.002, 0.04, 0.35, 0.35, 0.35])
  movel(T(p[0.195151, -0.310505, 0.050000, 3.14159, 0.0, 0.0]), a=A_DEFAULT*ACCEL_FACTOR, v=V_RECT*SPEED_FACTOR, r=0.002)
  movel(T(p[0.190303, -0.315354, 0.050000, 3.14159, 0.0, 0.0]), a=A_DEFAULT*ACCEL_FACTOR, v=V_RECT*SPEED_FACTOR, r=0.002)
  movel(T(p[0.185454, -0.320203, 0.050000, 3.14159, 0.0, 0.0]), a=A_DEFAULT*ACCEL_FACTOR, v=V_RECT*SPEED_FACTOR, r=0.002)
  movel(T(p[0.180605, -0.325052, 0.050000, 3.14159, 0.0, 0.0]), a=A_DEFAULT*ACCEL_FACTOR, v=V_RECT*SPEED_FACTOR, r=0.002)
  movel(T(p[0.175756, -0.329901, 0.050000, 3.14159, 0.0, 0.0]), a=A_DEFAULT*ACCEL_FACTOR, v=V_RECT*SPEED_FACTOR, r=0.002)
  movel(T(p[0.170908, -0.334749, 0.050000, 3.14159, 0.0, 0.0]), a=A_DEFAULT*ACCEL_FACTOR, v=V_RECT*SPEED_FACTOR, r=0.002)
  movel(T(p[0.176413, -0.334194, 0.050000, 3.14159, 0.0, 0.0]), a=A_DEFAULT*ACCEL_FACTOR, v=V_RECT*SPEED_FACTOR, r=0.002)
  movel(T(p[0.181262, -0.329345, 0.050000, 3.14159, 0.0, 0.0]), a=A_DEFAULT*ACCEL_FACTOR, v=V_RECT*SPEED_FACTOR, r=0.002)
  movel(T(p[0.186110, -0.324496, 0.050000, 3.14159, 0.0, 0.0]), a=A_DEFAULT*ACCEL_FACTOR, v=V_RECT*SPEED_FACTOR, r=0.002)
  movel(T(p[0.190959, -0.319648, 0.050000, 3.14159, 0.0, 0.0]), a=A_DEFAULT*ACCEL_FACTOR, v=V_RECT*SPEED_FACTOR, r=0.002)
  movel(T(p[0.195808, -0.314799, 0.050000, 3.14159, 0.0, 0.0]), a=A_DEFAULT*ACCEL_FACTOR, v=V_RECT*SPEED_FACTOR, r=0.002)
  movel(T(p[0.200657, -0.309950, 0.050000, 3.14159, 0.0, 0.0]), a=A_DEFAULT*ACCEL_FACTOR, v=V_RECT*SPEED_FACTOR, r=0.002)
  movel(T(p[0.202525, -0.313031, 0.050000, 3.14159, 0.0, 0.0]), a=A_DEFAULT*ACCEL_FACTOR, v=V_RECT*SPEED_FACTOR, r=0.002)
  movel(T(p[0.197676, -0.317880, 0.050000, 3.14159, 0.0, 0.0]), a=A_DEFAULT*ACCEL_FACTOR, v=V_RECT*SPEED_FACTOR, r=0.002)
  movel(T(p[0.192828, -0.322729, 0.050000, 3.14159, 0.0, 0.0]), a=A_DEFAULT*ACCEL_FACTOR, v=V_RECT*SPEED_FACTOR, r=0.002)
  movel(T(p[0.187979, -0.327577, 0.050000, 3.14159, 0.0, 0.0]), a=A_DEFAULT*ACCEL_FACTOR, v=V_RECT*SPEED_FACTOR, r=0.002)
  movel(T(p[0.183131, -0.332426, 0.050000, 3.14159, 0.0, 0.0]), a=A_DEFAULT*ACCEL_FACTOR, v=V_RECT*SPEED_FACTOR, r=0.002)
  movel(T(p[0.178282, -0.337274, 0.050000, 3.14159, 0.0, 0.0]), a=A_DEFAULT*ACCEL_FACTOR, v=V_RECT*SPEED_FACTOR, r=0.002)
  movel(T(p[0.178938, -0.341568, 0.050000, 3.14159, 0.0, 0.0]), a=A_DEFAULT*ACCEL_FACTOR, v=V_RECT*SPEED_FACTOR, r=0.002)
  movel(T(p[0.183787, -0.336719, 0.050000, 3.14159, 0.0, 0.0]), a=A_DEFAULT*ACCEL_FACTOR, v=V_RECT*SPEED_FACTOR, r=0.002)
  movel(T(p[0.188636, -0.331870, 0.050000, 3.14159, 0.0, 0.0]), a=A_DEFAULT*ACCEL_FACTOR, v=V_RECT*SPEED_FACTOR, r=0.002)
  movel(T(p[0.193485, -0.327021, 0.050000, 3.14159, 0.0, 0.0]), a=A_DEFAULT*ACCEL_FACTOR, v=V_RECT*SPEED_FACTOR, r=0.002)
  movel(T(p[0.198333, -0.322173, 0.050000, 3.14159, 0.0, 0.0]), a=A_DEFAULT*ACCEL_FACTOR, v=V_RECT*SPEED_FACTOR, r=0.002)
  movel(T(p[0.203182, -0.317324, 0.050000, 3.14159, 0.0, 0.0]), a=A_DEFAULT*ACCEL_FACTOR, v=V_RECT*SPEED_FACTOR, r=0.002)
  movel(T(p[0.209899, -0.315556, 0.050000, 3.14159, 0.0, 0.0]), a=A_DEFAULT*ACCEL_FACTOR, v=V_RECT*SPEED_FACTOR, r=0.002)
  movel(T(p[0.205051, -0.320405, 0.050000, 3.14159, 0.0, 0.0]), a=A_DEFAULT*ACCEL_FACTOR, v=V_RECT*SPEED_FACTOR, r=0.002)
  movel(T(p[0.200202, -0.325254, 0.050000, 3.14159, 0.0, 0.0]), a=A_DEFAULT*ACCEL_FACTOR, v=V_RECT*SPEED_FACTOR, r=0.002)
  movel(T(p[0.195354, -0.330102, 0.050000, 3.14159, 0.0, 0.0]), a=A_DEFAULT*ACCEL_FACTOR, v=V_RECT*SPEED_FACTOR, r=0.002)
  movel(T(p[0.190504, -0.334952, 0.050000, 3.14159, 0.0, 0.0]), a=A_DEFAULT*ACCEL_FACTOR, v=V_RECT*SPEED_FACTOR, r=0.002)
  movel(T(p[0.185656, -0.339800, 0.050000, 3.14159, 0.0, 0.0]), a=A_DEFAULT*ACCEL_FACTOR, v=V_RECT*SPEED_FACTOR, r=0.002)
  movel(T(p[0.180807, -0.344649, 0.050000, 3.14159, 0.0, 0.0]), a=A_DEFAULT*ACCEL_FACTOR, v=V_RECT*SPEED_FACTOR, r=0.002)
  movel(T(p[0.186313, -0.344093, 0.050000, 3.14159, 0.0, 0.0]), a=A_DEFAULT*ACCEL_FACTOR, v=V_RECT*SPEED_FACTOR, r=0.002)
  movel(T(p[0.191161, -0.339244, 0.050000, 3.14159, 0.0, 0.0]), a=A_DEFAULT*ACCEL_FACTOR, v=V_RECT*SPEED_FACTOR, r=0.002)
  movel(T(p[0.196010, -0.334396, 0.050000, 3.14159, 0.0, 0.0]), a=A_DEFAULT*ACCEL_FACTOR, v=V_RECT*SPEED_FACTOR, r=0.002)
  movel(T(p[0.200858, -0.329547, 0.050000, 3.14159, 0.0, 0.0]), a=A_DEFAULT*ACCEL_FACTOR, v=V_RECT*SPEED_FACTOR, r=0.002)
  movel(T(p[0.205707, -0.324699, 0.050000, 3.14159, 0.0, 0.0]), a=A_DEFAULT*ACCEL_FACTOR, v=V_RECT*SPEED_FACTOR, r=0.002)
  movel(T(p[0.210556, -0.319849, 0.050000, 3.14159, 0.0, 0.0]), a=A_DEFAULT*ACCEL_FACTOR, v=V_RECT*SPEED_FACTOR, r=0.002)
  movel(T(p[0.212425, -0.322931, 0.050000, 3.14159, 0.0, 0.0]), a=A_DEFAULT*ACCEL_FACTOR, v=V_RECT*SPEED_FACTOR, r=0.002)
  movel(T(p[0.207576, -0.327779, 0.050000, 3.14159, 0.0, 0.0]), a=A_DEFAULT*ACCEL_FACTOR, v=V_RECT*SPEED_FACTOR, r=0.002)
  movel(T(p[0.202727, -0.332628, 0.050000, 3.14159, 0.0, 0.0]), a=A_DEFAULT*ACCEL_FACTOR, v=V_RECT*SPEED_FACTOR, r=0.002)
  movel(T(p[0.197879, -0.337477, 0.050000, 3.14159, 0.0, 0.0]), a=A_DEFAULT*ACCEL_FACTOR, v=V_RECT*SPEED_FACTOR, r=0.002)
  movel(T(p[0.193030, -0.342325, 0.050000, 3.14159, 0.0, 0.0]), a=A_DEFAULT*ACCEL_FACTOR, v=V_RECT*SPEED_FACTOR, r=0.002)
  movel(T(p[0.188181, -0.347174, 0.050000, 3.14159, 0.0, 0.0]), a=A_DEFAULT*ACCEL_FACTOR, v=V_RECT*SPEED_FACTOR, r=0.002)
  movel(T(p[0.188838, -0.351467, 0.050000, 3.14159, 0.0, 0.0]), a=A_DEFAULT*ACCEL_FACTOR, v=V_RECT*SPEED_FACTOR, r=0.002)
  movel(T(p[0.193686, -0.346619, 0.050000, 3.14159, 0.0, 0.0]), a=A_DEFAULT*ACCEL_FACTOR, v=V_RECT*SPEED_FACTOR, r=0.002)
  movel(T(p[0.198536, -0.341770, 0.050000, 3.14159, 0.0, 0.0]), a=A_DEFAULT*ACCEL_FACTOR, v=V_RECT*SPEED_FACTOR, r=0.002)
  movel(T(p[0.203384, -0.336921, 0.050000, 3.14159, 0.0, 0.0]), a=A_DEFAULT*ACCEL_FACTOR, v=V_RECT*SPEED_FACTOR, r=0.002)
  movel(T(p[0.208233, -0.332072, 0.050000, 3.14159, 0.0, 0.0]), a=A_DEFAULT*ACCEL_FACTOR, v=V_RECT*SPEED_FACTOR, r=0.002)
  movel(T(p[0.213081, -0.327224, 0.050000, 3.14159, 0.0, 0.0]), a=A_DEFAULT*ACCEL_FACTOR, v=V_RECT*SPEED_FACTOR, r=0.002)
  movel(T(p[0.219799, -0.325456, 0.050000, 3.14159, 0.0, 0.0]), a=A_DEFAULT*ACCEL_FACTOR, v=V_RECT*SPEED_FACTOR, r=0.002)
  movel(T(p[0.214950, -0.330304, 0.050000, 3.14159, 0.0, 0.0]), a=A_DEFAULT*ACCEL_FACTOR, v=V_RECT*SPEED_FACTOR, r=0.002)
  movel(T(p[0.210102, -0.335153, 0.050000, 3.14159, 0.0, 0.0]), a=A_DEFAULT*ACCEL_FACTOR, v=V_RECT*SPEED_FACTOR, r=0.002)
  movel(T(p[0.205253, -0.340002, 0.050000, 3.14159, 0.0, 0.0]), a=A_DEFAULT*ACCEL_FACTOR, v=V_RECT*SPEED_FACTOR, r=0.002)
  movel(T(p[0.200404, -0.344851, 0.050000, 3.14159, 0.0, 0.0]), a=A_DEFAULT*ACCEL_FACTOR, v=V_RECT*SPEED_FACTOR, r=0.002)
  movel(T(p[0.195555, -0.349700, 0.050000, 3.14159, 0.0, 0.0]), a=A_DEFAULT*ACCEL_FACTOR, v=V_RECT*SPEED_FACTOR, r=0.002)
  movel(T(p[0.190706, -0.354548, 0.050000, 3.14159, 0.0, 0.0]), a=A_DEFAULT*ACCEL_FACTOR, v=V_RECT*SPEED_FACTOR, r=0.002)
  movel(T(p[0.196212, -0.353993, 0.050000, 3.14159, 0.0, 0.0]), a=A_DEFAULT*ACCEL_FACTOR, v=V_RECT*SPEED_FACTOR, r=0.002)
  movel(T(p[0.201061, -0.349144, 0.050000, 3.14159, 0.0, 0.0]), a=A_DEFAULT*ACCEL_FACTOR, v=V_RECT*SPEED_FACTOR, r=0.002)
  movel(T(p[0.205909, -0.344295, 0.050000, 3.14159, 0.0, 0.0]), a=A_DEFAULT*ACCEL_FACTOR, v=V_RECT*SPEED_FACTOR, r=0.002)
  movel(T(p[0.210758, -0.339447, 0.050000, 3.14159, 0.0, 0.0]), a=A_DEFAULT*ACCEL_FACTOR, v=V_RECT*SPEED_FACTOR, r=0.002)
  movel(T(p[0.215607, -0.334598, 0.050000, 3.14159, 0.0, 0.0]), a=A_DEFAULT*ACCEL_FACTOR, v=V_RECT*SPEED_FACTOR, r=0.002)
  movel(T(p[0.220456, -0.329749, 0.050000, 3.14159, 0.0, 0.0]), a=A_DEFAULT*ACCEL_FACTOR, v=V_RECT*SPEED_FACTOR, r=0.002)
  movel(T(p[0.222324, -0.332830, 0.050000, 3.14159, 0.0, 0.0]), a=A_DEFAULT*ACCEL_FACTOR, v=V_RECT*SPEED_FACTOR, r=0.002)
  movel(T(p[0.217475, -0.337679, 0.050000, 3.14159, 0.0, 0.0]), a=A_DEFAULT*ACCEL_FACTOR, v=V_RECT*SPEED_FACTOR, r=0.002)
  movel(T(p[0.212627, -0.342528, 0.050000, 3.14159, 0.0, 0.0]), a=A_DEFAULT*ACCEL_FACTOR, v=V_RECT*SPEED_FACTOR, r=0.002)
  movel(T(p[0.207778, -0.347376, 0.050000, 3.14159, 0.0, 0.0]), a=A_DEFAULT*ACCEL_FACTOR, v=V_RECT*SPEED_FACTOR, r=0.002)
  movel(T(p[0.202930, -0.352225, 0.050000, 3.14159, 0.0, 0.0]), a=A_DEFAULT*ACCEL_FACTOR, v=V_RECT*SPEED_FACTOR, r=0.002)
  movel(T(p[0.198081, -0.357073, 0.050000, 3.14159, 0.0, 0.0]), a=A_DEFAULT*ACCEL_FACTOR, v=V_RECT*SPEED_FACTOR, r=0.002)
  movel(T(p[0.198737, -0.361367, 0.050000, 3.14159, 0.0, 0.0]), a=A_DEFAULT*ACCEL_FACTOR, v=V_RECT*SPEED_FACTOR, r=0.002)
  movel(T(p[0.203586, -0.356518, 0.050000, 3.14159, 0.0, 0.0]), a=A_DEFAULT*ACCEL_FACTOR, v=V_RECT*SPEED_FACTOR, r=0.002)
  movel(T(p[0.208435, -0.351669, 0.050000, 3.14159, 0.0, 0.0]), a=A_DEFAULT*ACCEL_FACTOR, v=V_RECT*SPEED_FACTOR, r=0.002)
  movel(T(p[0.213284, -0.346820, 0.050000, 3.14159, 0.0, 0.0]), a=A_DEFAULT*ACCEL_FACTOR, v=V_RECT*SPEED_FACTOR, r=0.002)
  movel(T(p[0.218132, -0.341972, 0.050000, 3.14159, 0.0, 0.0]), a=A_DEFAULT*ACCEL_FACTOR, v=V_RECT*SPEED_FACTOR, r=0.002)
  movel(T(p[0.222981, -0.337123, 0.050000, 3.14159, 0.0, 0.0]), a=A_DEFAULT*ACCEL_FACTOR, v=V_RECT*SPEED_FACTOR, r=0.002)
  movel(T(p[0.229698, -0.335355, 0.050000, 3.14159, 0.0, 0.0]), a=A_DEFAULT*ACCEL_FACTOR, v=V_RECT*SPEED_FACTOR, r=0.002)
  movel(T(p[0.224850, -0.340204, 0.050000, 3.14159, 0.0, 0.0]), a=A_DEFAULT*ACCEL_FACTOR, v=V_RECT*SPEED_FACTOR, r=0.002)
  movel(T(p[0.220001, -0.345053, 0.050000, 3.14159, 0.0, 0.0]), a=A_DEFAULT*ACCEL_FACTOR, v=V_RECT*SPEED_FACTOR, r=0.002)
  movel(T(p[0.215153, -0.349901, 0.050000, 3.14159, 0.0, 0.0]), a=A_DEFAULT*ACCEL_FACTOR, v=V_RECT*SPEED_FACTOR, r=0.002)
  movel(T(p[0.210303, -0.354751, 0.050000, 3.14159, 0.0, 0.0]), a=A_DEFAULT*ACCEL_FACTOR, v=V_RECT*SPEED_FACTOR, r=0.002)
  movel(T(p[0.205455, -0.359599, 0.050000, 3.14159, 0.0, 0.0]), a=A_DEFAULT*ACCEL_FACTOR, v=V_RECT*SPEED_FACTOR, r=0.002)
  movel(T(p[0.200606, -0.364448, 0.050000, 3.14159, 0.0, 0.0]), a=A_DEFAULT*ACCEL_FACTOR, v=V_RECT*SPEED_FACTOR, r=0.002)
  end_force_mode()
  movel(T(p[0.200000, -0.365054, 0.060000, 3.14159, 0.0, 0.0]), a=A_DEFAULT*ACCEL_FACTOR, v=V_APPROACH*SPEED_FACTOR)
end

def etalement():
  set_tcp(p[0.0, 0.0, 0.072, 0, 0, 0])
  movej(T(p[0.2, -0.3, 0.060000, 3.14159, 0.0, 0.0]), a=A_INIT*ACCEL_FACTOR, v=V_INIT*SPEED_FACTOR)

  cycle_1()
  cycle_2()
  cycle_3()
  cycle_4()
  cycle_5()
  cycle_6()
end

etalement()
